// TIA Portal V19 export
FUNCTION_BLOCK "AccRollConveyor_FB"   // FB162, LAD
TITLE = Acc roll conveyor
// stored: MemoryReserve 100, SetENOAutomatically false
   VAR_INPUT
      AreaInterface : "AreaInterface";
      ZSI : "udt_ZoneSafetyInterface";
      DSI : Struct
         Roll1 : "udt_DeviceSafetyInterface";
         Roll2 : "udt_DeviceSafetyInterface";
         Roll3 : "udt_DeviceSafetyInterface";
         PusherVert : "udt_DeviceSafetyInterface";
         PusherHoriz : "udt_DeviceSafetyInterface";
      END_STRUCT;
      Drive : Struct
         Roll1 : "TAx_DriveInterface";
         Roll2 : "TAx_DriveInterface";
         Roll3 : "TAx_DriveInterface";
      END_STRUCT;
      HWID : Struct
         Roll1_TEL1 : HW_SUBMODULE;
         Roll2_TEL1 : HW_SUBMODULE;
         Roll3_TEL1 : HW_SUBMODULE;
      END_STRUCT;
      DataIn : Struct
         Pb_Semiauto : Bool;
         Rolls_PbFwd : Bool;
         Rolls_PbBwd : Bool;
         PusherVert_PbUp : Bool;
         PusherVert_PbDown : Bool;
         PusherHoriz_PbLeft : Bool;
         PusherHoriz_PbRight : Bool;
         SensorMatPresence_S2_Entry : Bool;
         SensorMatPresence_S3 : Bool;
         SensorMatPresence_S4 : Bool;
         SensorMatPresence_S5_Stop : Bool;
         ExitLeft_MatPresence1 : Bool;
         ExitLeft_MatPresence2 : Bool;
         ExitLeft_MatPresence3 : Bool;
         ExitLeft_MatPresence4 : Bool;
      END_STRUCT;
      CIn : Struct
         Manager : Struct
            EnableStopDoorOpeningReq : Bool;
            EnableStopInPhase : Bool;
            EnableStopProgrammed : Bool;
         END_STRUCT;
         Semiautomatic : Bool;
         A03_CanLoadPiece : Bool;
         A03_InCycle : Bool;
         ReqFwdFromCut : Bool;
         StopCheckQuality : Bool;
      END_STRUCT;
      Config : Struct
         Roll1 : "SpeedMachine_Config";
         Roll2 : "SpeedMachine_Config";
         Roll3 : "SpeedMachine_Config";
         PusherVert : Array[1..6] of "ValveMachine_Config";
         PusherHoriz : Array[1..6] of "ValveMachine_Config";
         SensorsDelayOn : Time := T#100ms;
         SensorsDelayOff : Time := T#100ms;
         ExitLeftDelayOn : Time := T#100ms;
         ExitLeftDelayOff : Time := T#100ms;
      END_STRUCT;
   END_VAR
   VAR_OUTPUT
      MachineInterface : "MachineInterface";
      COut : Struct
         Rolls : Struct
            Infeed_ReqON : Bool;
            Bwd_CheckNext : Bool;
            Fwd_CheckNext : Bool;
            Standstill : Bool;
         END_STRUCT;
         PusherVert : Struct
            Rest_CheckNext : Bool;
            Work_CheckNext : Bool;
            AllStandstill : Bool;
            TwoUp : Bool;
            AllDown : Bool;
         END_STRUCT;
         PusherHoriz : Struct
            Left_CheckNext : Bool;
            Right_CheckNext : Bool;
            AllStandstill : Bool;
            InLeftPos : Bool;
            InRightPos : Bool;
         END_STRUCT;
         Manager : "udt_AccRollConveyor_COut_Manager";
      END_STRUCT;
   END_VAR
   VAR_IN_OUT
      Pers : "udt_AccRollConveyor_Pers";
   END_VAR
   VAR
      Sts : Struct
         Semiautomatic : Bool;
         OP_CanMoveFreely : Bool;
         NextTargetPathLeft : Bool;
         NextTargetPathRight : Bool;
         ActTargetPathLeft : Bool;
         ActTargetPathRight : Bool;
         TrkExitLeftFull : Bool;
         TrkPieceInRolls : Int;
         TrkPieceToCheckInRoll : Int;
         TrkPieceInLenght : LReal;
         TrkPieceRecondGoodFind : Int;
         StopCutCheckPiece : Bool;
         Pusher : Struct
            InLeftPos : Bool;
            InRightPos : Bool;
            UsedInLeftPos : Bool;
            UsedInRightPos : Bool;
            AllDown : Bool;
            TwoUp : Bool;
            Used : Array[1.."MAX_PUSHER"] of Bool;
         END_STRUCT;
         CycleTime : Struct
            PusherHoriz : Struct
               DT_W_Start : DTL;
               DT_W_Stop : DTL;
               DT_R_Start : DTL;
               DT_R_Stop : DTL;
               R_To_W_Exe : Bool;
               W_To_R_Exe : Bool;
               R_To_W_Items : Int;
               R_To_W_Sum : Time;
               W_To_R_Items : Int;
               W_To_R_Sum : Time;
            END_STRUCT;
            PPrf_PrgNoSave : DInt;
         END_STRUCT;
      END_STRUCT;
      Ctrl : Struct
         StopInPhase : Bool;
         StopProgrammed : Bool;
         Pb_Semiauto : Bool;
         Rolls : Struct
            Man_Fwd : Bool;
            Man_Bwd : Bool;
            Aut_SlowDown : Bool;
            Aut_Fwd : Bool;
            Vel : LReal;
            Entry_Vel : LReal;
            Acc : LReal;
            Dec : LReal;
         END_STRUCT;
         Pusher : Struct
            Man_Left : Bool;
            Man_Right : Bool;
            Man_Up : Bool;
            Man_Down : Bool;
            Aut_Left : Bool;
            Aut_Right : Bool;
            Aut_Up : Bool;
            Aut_Down : Bool;
         END_STRUCT;
         Cycle : Struct
            ReqNextMovePieceToLeft : Bool;
            ReqNextMovePieceToRight : Bool;
            ExeNextMovePieceToLeft : Bool;
            ExeNextMovePieceToRight : Bool;
            ReqMovePieceToLeft : Bool;
            ReqMovePieceToRight : Bool;
            ExeMovePieceToLeft : Bool;
            ExeMovePieceToRight : Bool;
         END_STRUCT;
      END_STRUCT;
      Alarm : Struct
         Roll1 : "SpeedMachine_Alr";
         Roll2 : "SpeedMachine_Alr";
         Roll3 : "SpeedMachine_Alr";
         PusherVert : Array[1.."MAX_PUSHER"] of "ValveAlr";
         PusherHoriz : Array[1.."MAX_PUSHER"] of "ValveAlr";
         TrkCloggedLeftExit : Bool;
         TrkCloggedRightA03 : Bool;
         TrkCloggedRollway : Bool;
         TrkWrongMismatch_P0 : Bool;
         TrkExitFullToChek : Bool;
      END_STRUCT;
      Warning : Struct
         Roll1 : "SpeedMachine_Wng";
         Roll2 : "SpeedMachine_Wng";
         Roll3 : "SpeedMachine_Wng";
         PusherVert : Array[1.."MAX_PUSHER"] of "ValveMachine_Wng";
         PusherHoriz : Array[1.."MAX_PUSHER"] of "ValveMachine_Wng";
      END_STRUCT;
      HMI : Struct
         PusherHoriz : Struct
            Last_R_to_W_ID : DInt;
            Last_R_to_W_Time : Time;
            Last_W_to_R_ID : DInt;
            Last_W_to_R_Time : Time;
            Avg_R_to_W_Time : Time;
            Avg_W_to_R_Time : Time;
            Avg_CycleTime_S : LReal;
            Buffer_R_to_W_Time : Array[1..#BUFFER_ITEMS] of Struct
               ID : DInt;
               Value : Time;
            END_STRUCT;
            Buffer_W_to_R_Time : Array[1..#BUFFER_ITEMS] of Struct
               ID : DInt;
               Value : Time;
            END_STRUCT;
         END_STRUCT;
      END_STRUCT;
      Roll1 : "SpeedMachine_FB";
      Roll2 : "SpeedMachine_FB";
      Roll3 : "SpeedMachine_FB";
      PusherVert : Array[1.."MAX_PUSHER"] of "ValveMachine_FB";
      PusherHoriz : Array[1.."MAX_PUSHER"] of "ValveMachine_FB";
      MatPresence_S2_Entry : "DelayOnOff_R";
      MatPresence_S3 : "DelayOnOff_R";
      MatPresence_S4 : "DelayOnOff_R";
      MatPresence_S5_Stop : "DelayOnOff_R";
      MatPresence_ExitLeft1 : "DelayOnOff_R";
      MatPresence_ExitLeft2 : "DelayOnOff_R";
      MatPresence_ExitLeft3 : "DelayOnOff_R";
      MatPresence_ExitLeft4 : "DelayOnOff_R";
      tonSlowDownRolls { S7_SetPoint := 'True'} : TON_TIME;
      tonStopRollformer : TON_TIME;
      tonSlowDownRollformer : TON_TIME;
      tonTrkMismatcP0 { S7_SetPoint := 'True'} : TON_TIME;
      Rollway_Control : "Rulliera_Control_FB";
      AUX : Struct
         Pb_Semiauto { ExternalAccessible := 'False'; ExternalVisible := 'False'; ExternalWritable := 'False'} : Bool;
         Rolls_PbFwd : Bool;
         Rolls_PbBwd : Bool;
         PusherVert_PbUp : Bool;
         PusherVert_PbDopwn : Bool;
         PusherHoriz_PbLeft : Bool;
         PusherHoriz_PbRight : Bool;
         NE_MatPresence2_Entry { ExternalAccessible := 'False'; ExternalVisible := 'False'; ExternalWritable := 'False'} : Bool;
         PE_MatPresence3 : Bool;
         PE_MatPresence5_Stop : Bool;
         PE_SlowDownRolls : Bool;
         NE_SlowDownDone : Bool;
         PusherHoriz_InLeftPos : Bool;
         PusherHoriz_InRightPos : Bool;
      END_STRUCT;
      PusherVert_MachineInterface { ExternalAccessible := 'False'; ExternalVisible := 'False'; ExternalWritable := 'False'} : "MachineInterface";
      PusherHoriz_MachineInterface { ExternalAccessible := 'False'; ExternalVisible := 'False'; ExternalWritable := 'False'} : "MachineInterface";
   END_VAR
   VAR_TEMP
      PE : Struct
         Pb_Semiauto : Bool;
         Rolls_PbFwd : Bool;
         Rolls_PbBwd : Bool;
         PusherVert_PbUp : Bool;
         PusherVert_PbDown : Bool;
         PusherHoriz_PbLeft : Bool;
         PusherHoriz_PbRight : Bool;
         NE_MatPresence2_Entry : Bool;
         PE_MatPresence3 : Bool;
         PE_MatPresence5_Stop : Bool;
         PE_SlowDownRolls : Bool;
         NE_SlowDownDone : Bool;
         PusherHoriz_InLeftPos : Bool;
         PusherHoriz_InRightPos : Bool;
      END_STRUCT;
      i : Int;
      PusherVert_NrUp : Int;
      ActualPieceLenght : LReal;
      RetVal_MOVEBLK : Int;
      Ptrk_ItemFind : Int;
      Ptrk_ExitItemToCheck : Int;
      ReturnVal : Word;
      AddAlarm : Bool;
      PartLenght : LReal;
   END_VAR
   VAR CONSTANT
      BUFFER_ITEMS : Int := 10;
   END_VAR
   VAR_TEMP   // added for the SCL form of the ladder/FBD networks
      _w1 : Bool;
      _w2 : Bool;
      _w3 : Bool;
      _w4 : Bool;
      _w5 : Bool;
   END_VAR
BEGIN

REGION Network 1 (SCL): Reset alarms command

   IF  #AreaInterface.RstAlarms THEN
       // Alarms
       #Alarm.TrkCloggedLeftExit := FALSE;
       #Alarm.TrkCloggedRightA03 := FALSE;
       #Alarm.TrkCloggedRollway := FALSE;

       #Alarm.TrkWrongMismatch_P0 := FALSE;
       #Alarm.TrkExitFullToChek := FALSE;

   END_IF;
END_REGION

REGION Network 2: >
END_REGION

REGION Network 3: OP Can move freely
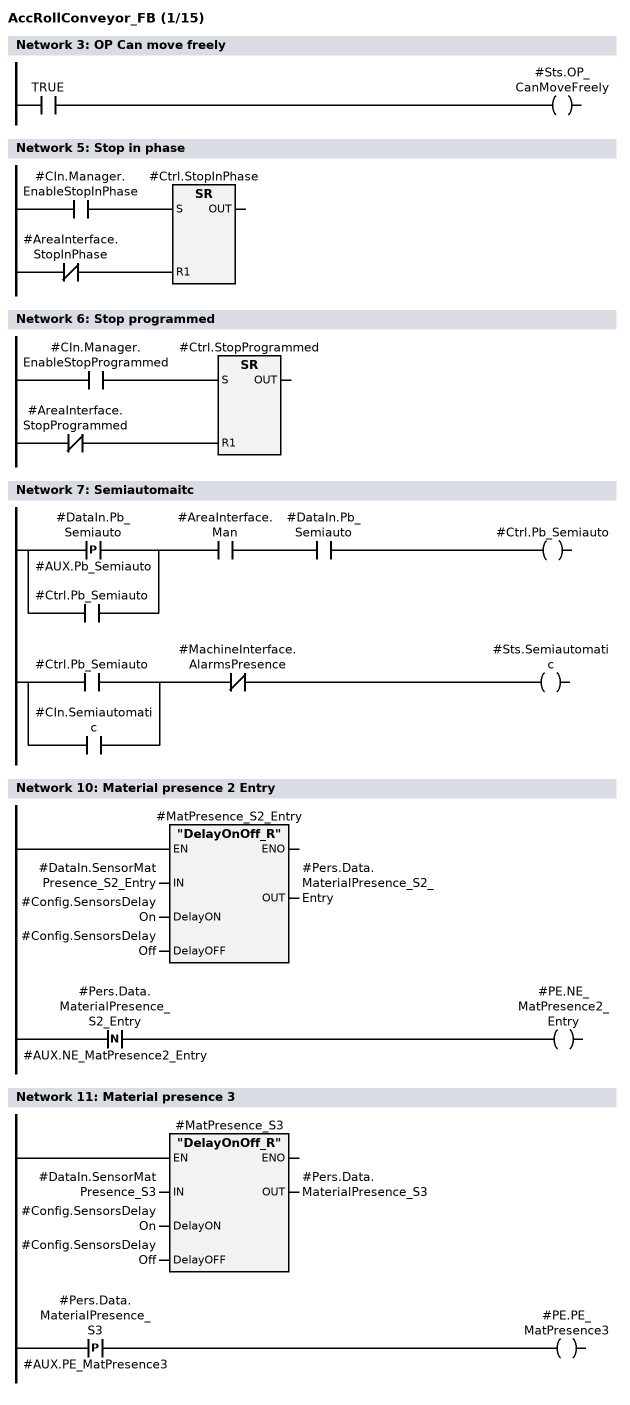
   RUNG wire#powerrail
      Contact( TRUE )
      Coil( #Sts.OP_CanMoveFreely )
   END_RUNG
   // the same network as SCL:
   #Sts.OP_CanMoveFreely := TRUE;
END_REGION

REGION Network 5: Stop in phase
   RUNG wire#powerrail
      Contact( #CIn.Manager.EnableStopInPhase )
      S_SR(operand := #Ctrl.StopInPhase, r1 := wire#w1)
   END_RUNG
   RUNG wire#powerrail
      I_Contact( #AreaInterface.StopInPhase )
   END_RUNG wire#w1
   // the same network as SCL:
   IF #CIn.Manager.EnableStopInPhase THEN
       #Ctrl.StopInPhase := TRUE;   // SR flip-flop
   END_IF;
   IF NOT #AreaInterface.StopInPhase THEN #Ctrl.StopInPhase := FALSE; END_IF;
END_REGION

REGION Network 6: Stop programmed
   RUNG wire#powerrail
      Contact( #CIn.Manager.EnableStopProgrammed )
      S_SR(operand := #Ctrl.StopProgrammed, r1 := wire#w1)
   END_RUNG
   RUNG wire#powerrail
      I_Contact( #AreaInterface.StopProgrammed )
   END_RUNG wire#w1
   // the same network as SCL:
   IF #CIn.Manager.EnableStopProgrammed THEN
       #Ctrl.StopProgrammed := TRUE;   // SR flip-flop
   END_IF;
   IF NOT #AreaInterface.StopProgrammed THEN #Ctrl.StopProgrammed := FALSE; END_IF;
END_REGION

REGION Network 7: Semiautomaitc
   RUNG wire#powerrail
      P_Contact(operand := #DataIn.Pb_Semiauto, bit := #AUX.Pb_Semiauto)
      wire#w1
      Contact( #AreaInterface.Man )
      Contact( #DataIn.Pb_Semiauto )
      Coil( #Ctrl.Pb_Semiauto )
   END_RUNG
   RUNG wire#powerrail
      Contact( #Ctrl.Pb_Semiauto )
   END_RUNG wire#w1
   RUNG wire#powerrail
      Contact( #Ctrl.Pb_Semiauto )
      wire#w2
      I_Contact( #MachineInterface.AlarmsPresence )
      Coil( #Sts.Semiautomatic )
   END_RUNG
   RUNG wire#powerrail
      Contact( #CIn.Semiautomatic )
   END_RUNG wire#w2
   // the same network as SCL:
   #_w1 := #DataIn.Pb_Semiauto AND NOT #AUX.Pb_Semiauto;   // rising edge of #DataIn.Pb_Semiauto
   #AUX.Pb_Semiauto := #DataIn.Pb_Semiauto;
   #Ctrl.Pb_Semiauto := (#_w1 OR #Ctrl.Pb_Semiauto) AND #AreaInterface.Man AND #DataIn.Pb_Semiauto;
   #Sts.Semiautomatic := (#Ctrl.Pb_Semiauto OR #CIn.Semiautomatic) AND NOT #MachineInterface.AlarmsPresence;
END_REGION

REGION Network 9: <<< SENSOR MAT PRESENCE >>>
END_REGION

REGION Network 10: Material presence 2 Entry
   RUNG wire#powerrail
      #MatPresence_S2_Entry(IN := #DataIn.SensorMatPresence_S2_Entry, DelayON := #Config.SensorsDelayOn, DelayOFF := #Config.SensorsDelayOff, OUT => #Pers.Data.MaterialPresence_S2_Entry)
   END_RUNG
   RUNG wire#powerrail
      N_Contact(operand := #Pers.Data.MaterialPresence_S2_Entry, bit := #AUX.NE_MatPresence2_Entry)
      Coil( #PE.NE_MatPresence2_Entry )
   END_RUNG
   // the same network as SCL:
   #MatPresence_S2_Entry(IN := #DataIn.SensorMatPresence_S2_Entry,   // "DelayOnOff_R"
                         DelayON := #Config.SensorsDelayOn,
                         DelayOFF := #Config.SensorsDelayOff,
                         OUT => #Pers.Data.MaterialPresence_S2_Entry);
   #_w1 := NOT #Pers.Data.MaterialPresence_S2_Entry AND #AUX.NE_MatPresence2_Entry;   // falling edge of #Pers.Data.MaterialPresence_S2_Entry
   #AUX.NE_MatPresence2_Entry := #Pers.Data.MaterialPresence_S2_Entry;
   #PE.NE_MatPresence2_Entry := #_w1;
END_REGION

REGION Network 11: Material presence 3
   RUNG wire#powerrail
      #MatPresence_S3(IN := #DataIn.SensorMatPresence_S3, DelayON := #Config.SensorsDelayOn, DelayOFF := #Config.SensorsDelayOff, OUT => #Pers.Data.MaterialPresence_S3)
   END_RUNG
   RUNG wire#powerrail
      P_Contact(operand := #Pers.Data.MaterialPresence_S3, bit := #AUX.PE_MatPresence3)
      Coil( #PE.PE_MatPresence3 )
   END_RUNG
   // the same network as SCL:
   #MatPresence_S3(IN := #DataIn.SensorMatPresence_S3,   // "DelayOnOff_R"
                   DelayON := #Config.SensorsDelayOn,
                   DelayOFF := #Config.SensorsDelayOff,
                   OUT => #Pers.Data.MaterialPresence_S3);
   #_w1 := #Pers.Data.MaterialPresence_S3 AND NOT #AUX.PE_MatPresence3;   // rising edge of #Pers.Data.MaterialPresence_S3
   #AUX.PE_MatPresence3 := #Pers.Data.MaterialPresence_S3;
   #PE.PE_MatPresence3 := #_w1;
END_REGION

REGION Network 12: Material presence 4
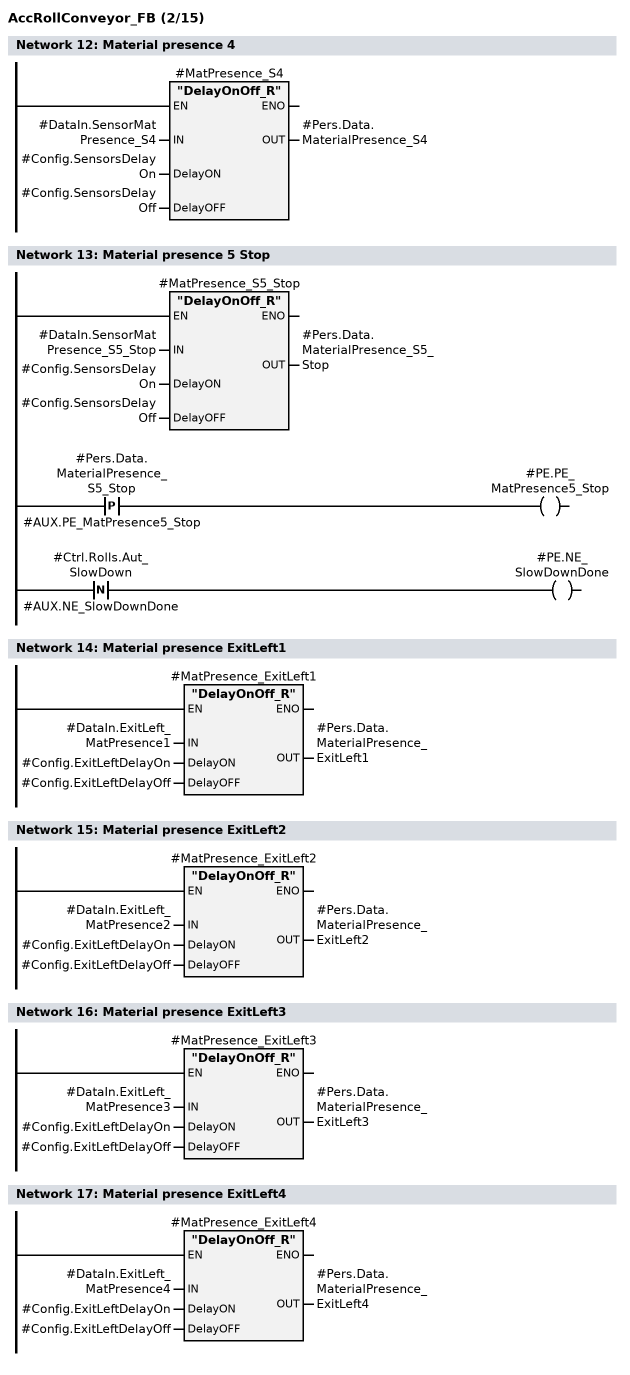
   RUNG wire#powerrail
      #MatPresence_S4(IN := #DataIn.SensorMatPresence_S4, DelayON := #Config.SensorsDelayOn, DelayOFF := #Config.SensorsDelayOff, OUT => #Pers.Data.MaterialPresence_S4)
   END_RUNG
   // the same network as SCL:
   #MatPresence_S4(IN := #DataIn.SensorMatPresence_S4,   // "DelayOnOff_R"
                   DelayON := #Config.SensorsDelayOn,
                   DelayOFF := #Config.SensorsDelayOff,
                   OUT => #Pers.Data.MaterialPresence_S4);
END_REGION

REGION Network 13: Material presence 5 Stop
   RUNG wire#powerrail
      #MatPresence_S5_Stop(IN := #DataIn.SensorMatPresence_S5_Stop, DelayON := #Config.SensorsDelayOn, DelayOFF := #Config.SensorsDelayOff, OUT => #Pers.Data.MaterialPresence_S5_Stop)
   END_RUNG
   RUNG wire#powerrail
      P_Contact(operand := #Pers.Data.MaterialPresence_S5_Stop, bit := #AUX.PE_MatPresence5_Stop)
      Coil( #PE.PE_MatPresence5_Stop )
   END_RUNG
   RUNG wire#powerrail
      N_Contact(operand := #Ctrl.Rolls.Aut_SlowDown, bit := #AUX.NE_SlowDownDone)
      Coil( #PE.NE_SlowDownDone )
   END_RUNG
   // the same network as SCL:
   #MatPresence_S5_Stop(IN := #DataIn.SensorMatPresence_S5_Stop,   // "DelayOnOff_R"
                        DelayON := #Config.SensorsDelayOn,
                        DelayOFF := #Config.SensorsDelayOff,
                        OUT => #Pers.Data.MaterialPresence_S5_Stop);
   #_w1 := #Pers.Data.MaterialPresence_S5_Stop AND NOT #AUX.PE_MatPresence5_Stop;   // rising edge of #Pers.Data.MaterialPresence_S5_Stop
   #AUX.PE_MatPresence5_Stop := #Pers.Data.MaterialPresence_S5_Stop;
   #PE.PE_MatPresence5_Stop := #_w1;
   #_w2 := NOT #Ctrl.Rolls.Aut_SlowDown AND #AUX.NE_SlowDownDone;   // falling edge of #Ctrl.Rolls.Aut_SlowDown
   #AUX.NE_SlowDownDone := #Ctrl.Rolls.Aut_SlowDown;
   #PE.NE_SlowDownDone := #_w2;
END_REGION

REGION Network 14: Material presence ExitLeft1
   RUNG wire#powerrail
      #MatPresence_ExitLeft1(IN := #DataIn.ExitLeft_MatPresence1, DelayON := #Config.ExitLeftDelayOn, DelayOFF := #Config.ExitLeftDelayOff, OUT => #Pers.Data.MaterialPresence_ExitLeft1)
   END_RUNG
   // the same network as SCL:
   #MatPresence_ExitLeft1(IN := #DataIn.ExitLeft_MatPresence1,   // "DelayOnOff_R"
                          DelayON := #Config.ExitLeftDelayOn,
                          DelayOFF := #Config.ExitLeftDelayOff,
                          OUT => #Pers.Data.MaterialPresence_ExitLeft1);
END_REGION

REGION Network 15: Material presence ExitLeft2
   RUNG wire#powerrail
      #MatPresence_ExitLeft2(IN := #DataIn.ExitLeft_MatPresence2, DelayON := #Config.ExitLeftDelayOn, DelayOFF := #Config.ExitLeftDelayOff, OUT => #Pers.Data.MaterialPresence_ExitLeft2)
   END_RUNG
   // the same network as SCL:
   #MatPresence_ExitLeft2(IN := #DataIn.ExitLeft_MatPresence2,   // "DelayOnOff_R"
                          DelayON := #Config.ExitLeftDelayOn,
                          DelayOFF := #Config.ExitLeftDelayOff,
                          OUT => #Pers.Data.MaterialPresence_ExitLeft2);
END_REGION

REGION Network 16: Material presence ExitLeft3
   RUNG wire#powerrail
      #MatPresence_ExitLeft3(IN := #DataIn.ExitLeft_MatPresence3, DelayON := #Config.ExitLeftDelayOn, DelayOFF := #Config.ExitLeftDelayOff, OUT => #Pers.Data.MaterialPresence_ExitLeft3)
   END_RUNG
   // the same network as SCL:
   #MatPresence_ExitLeft3(IN := #DataIn.ExitLeft_MatPresence3,   // "DelayOnOff_R"
                          DelayON := #Config.ExitLeftDelayOn,
                          DelayOFF := #Config.ExitLeftDelayOff,
                          OUT => #Pers.Data.MaterialPresence_ExitLeft3);
END_REGION

REGION Network 17: Material presence ExitLeft4
   RUNG wire#powerrail
      #MatPresence_ExitLeft4(IN := #DataIn.ExitLeft_MatPresence4, DelayON := #Config.ExitLeftDelayOn, DelayOFF := #Config.ExitLeftDelayOff, OUT => #Pers.Data.MaterialPresence_ExitLeft4)
   END_RUNG
   // the same network as SCL:
   #MatPresence_ExitLeft4(IN := #DataIn.ExitLeft_MatPresence4,   // "DelayOnOff_R"
                          DelayON := #Config.ExitLeftDelayOn,
                          DelayOFF := #Config.ExitLeftDelayOff,
                          OUT => #Pers.Data.MaterialPresence_ExitLeft4);
END_REGION

REGION Network 18: >
END_REGION

REGION Network 19: <<< TRACKING >>>
END_REGION

REGION Network 20 (SCL): Rollway movement

   //Tracking ENTRY to P6 
   IF "PTrk".A0202.P[PTRK_A0202_ENTRY].P_ID <> 0 AND
       ((#PE.NE_MatPresence2_Entry AND "PTrk".A0202.P[PTRK_A0202_ENTRY].PLen_Meas <= 4000) OR
       (#Pers.Data.MaterialPresence_S3 AND "PTrk".A0202.P[PTRK_A0202_ENTRY].PLen_Meas > 4000))
   THEN
       IF "PTrk".A0202.P[PTRK_A0202_P6].P_ID = 0 THEN
           "PTrk".A0202.P[PTRK_A0202_P6] := "PTrk".A0202.P[PTRK_A0202_ENTRY];
           "PTrk".A0202.P[PTRK_A0202_ENTRY] := "PTrk".Empty;
       ELSE
           #Alarm.TrkCloggedRollway := TRUE;
       END_IF;

   END_IF;


   //Sposto buffer tacking
   #i := "PTRK_A0202_P1";
   WHILE #i > "PTRK_A0202_P6" DO

       IF "PTrk".A0202.P[#i].P_ID = 0 AND
           "PTrk".A0202.P[#i - 1].P_ID <> 0
       THEN
           "PTrk".A0202.P[#i] := "PTrk".A0202.P[#i - 1];
           "PTrk".A0202.P[#i - 1] := "PTrk".Empty;
       END_IF;
       #i -= 1;

   END_WHILE;


   //Tracking P1 to P0
   IF "PTrk".A0202.P[PTRK_A0202_P1].P_ID <> 0 AND
       ((#PE.PE_MatPresence5_Stop AND #AreaInterface.Man AND NOT #Sts.Semiautomatic)
         OR #PE.NE_SlowDownDone)
   THEN
       IF "PTrk".A0202.P[PTRK_A0202_P0].P_ID = 0 THEN
           "PTrk".A0202.P[PTRK_A0202_P0] := "PTrk".A0202.P[PTRK_A0202_P1];
           "PTrk".A0202.P[PTRK_A0202_P1] := "PTrk".Empty;
       ELSE
           #Alarm.TrkCloggedRollway := TRUE;
       END_IF;
   END_IF;
END_REGION

REGION Network 21 (SCL): Left Exit movement

   //Rollway to left
   IF "PTrk".A0202.P[PTRK_A0202_P0].P_ID <> 0 AND
       (#Ctrl.Cycle.ReqMovePieceToLeft OR #AreaInterface.Man) AND
       #COut.PusherHoriz.Left_CheckNext AND NOT #COut.PusherHoriz.AllStandstill AND
       #Sts.Pusher.TwoUp AND
       NOT #Sts.Pusher.InLeftPos
   THEN

       IF "PTrk".A0202.P[PTRK_A0202_DEVITATOR_To_EXIT].P_ID = 0  THEN
           "PTrk".A0202.P[PTRK_A0202_DEVITATOR_To_EXIT] := "PTrk".A0202.P[PTRK_A0202_P0];
           "PTrk".A0202.P[PTRK_A0202_P0] := "PTrk".Empty;
       ELSE
           #Alarm.TrkCloggedLeftExit := TRUE;
       END_IF;
   END_IF;

   //Left to Exit
   IF "PTrk".A0202.P[PTRK_A0202_DEVITATOR_To_EXIT].P_ID <> 0 AND
       #Sts.Pusher.TwoUp AND
       #Sts.Pusher.UsedInLeftPos
   THEN

       #RetVal_MOVEBLK := MOVE_BLK_VARIANT(SRC := "PTrk".A02_EXIT_TOCHECK,
                                           COUNT := INT_TO_UDINT("PTRK_A0202_EXIT_TOCHECK_ITEMS" - 1),
                                           SRC_INDEX := 0,
                                           DEST_INDEX := 1,
                                           DEST => "PTrk".A02_EXIT_TOCHECK);

       "PTrk".A02_EXIT_TOCHECK[1] := "PTrk".A0202.P[PTRK_A0202_DEVITATOR_To_EXIT];
       "PTrk".A0202.P[PTRK_A0202_DEVITATOR_To_EXIT] := "PTrk".Empty;
   END_IF;

   //Alarm Clogged
   IF "PTrk".A0202.P[PTRK_A0202_DEVITATOR_To_EXIT].P_ID <> 0 AND
        "PTrk".A0202.P[PTRK_A0202_P0].P_ID <> 0
   THEN
       #Alarm.TrkCloggedLeftExit := TRUE;
   END_IF;
END_REGION

REGION Network 22 (SCL): Right A03 movement

   //Rollway to left
   IF "PTrk".A0202.P[PTRK_A0202_P0].P_ID <> 0 AND
       (#Ctrl.Cycle.ReqMovePieceToRight OR #AreaInterface.Man) AND
       #COut.PusherHoriz.Right_CheckNext AND NOT #COut.PusherHoriz.AllStandstill AND
       #Sts.Pusher.TwoUp AND 
       NOT #Sts.Pusher.InRightPos
   THEN

       IF "PTrk".A0202.P[PTRK_A0202_DEVIATOR_To_A0301].P_ID = 0 AND
           "PTrk".A0301.P[PTRK_A0301_Pos1_Entry].P_ID = 0
       THEN
           "PTrk".A0202.P[PTRK_A0202_DEVIATOR_To_A0301] := "PTrk".A0202.P[PTRK_A0202_P0];
           "PTrk".A0202.P[PTRK_A0202_P0] := "PTrk".Empty;
       ELSE
           #Alarm.TrkCloggedRightA03 := TRUE;
       END_IF;
   END_IF;

   //Left to Exit
   IF "PTrk".A0202.P[PTRK_A0202_DEVIATOR_To_A0301].P_ID <> 0 AND
       #Sts.Pusher.TwoUp AND
       #Sts.Pusher.UsedInRightPos
   THEN
       "PTrk".A0301.P[PTRK_A0301_Pos1_Entry] := "PTrk".A0202.P[PTRK_A0202_DEVIATOR_To_A0301];
       "PTrk".A0202.P[PTRK_A0202_DEVIATOR_To_A0301] := "PTrk".Empty;
   END_IF;

   //Alarm Clogged
   IF "PTrk".A0202.P[PTRK_A0202_DEVIATOR_To_A0301].P_ID <> 0 AND
       ("PTrk".A0301.P[PTRK_A0301_Pos1_Entry].P_ID <> 0 OR "PTrk".A0202.P[PTRK_A0202_P0].P_ID <> 0)
   THEN
       #Alarm.TrkCloggedRightA03 := TRUE;
   END_IF;
END_REGION

REGION Network 23 (SCL): Exit To check manager

   //Shift verso alto se trovo buco

   #Ptrk_ItemFind := 0;
   FOR #i := 1 TO "PTRK_A0202_EXIT_TOCHECK_ITEMS" - 1 DO

       IF "PTrk".A02_EXIT_TOCHECK[#i].P_ID = 0 AND
           "PTrk".A02_EXIT_TOCHECK[#i + 1].P_ID <> 0 THEN
           #Ptrk_ItemFind := #i;
           EXIT;
       END_IF;
   END_FOR;

   IF #Ptrk_ItemFind > 0 THEN
       #RetVal_MOVEBLK := MOVE_BLK_VARIANT(SRC := "PTrk".A02_EXIT_TOCHECK,
                                           COUNT := INT_TO_UDINT("PTRK_A0202_EXIT_TOCHECK_ITEMS" - #Ptrk_ItemFind),
                                           SRC_INDEX := #Ptrk_ItemFind,
                                           DEST_INDEX := #Ptrk_ItemFind - 1,
                                           DEST => "PTrk".A02_EXIT_TOCHECK);
   END_IF;



   //Conteggio Pezzi su rulliera
   #Sts.TrkPieceInRolls := 0;
   #Sts.TrkPieceInLenght := 0.0;
   #Sts.TrkPieceToCheckInRoll := 0;

   FOR #i := 1 TO "PTRK_A0202_DEVITATOR_To_EXIT" DO

       IF "PTrk".A0202.P[#i].P_ID <> 0 THEN
           #Sts.TrkPieceInRolls += 1;
           #Sts.TrkPieceInLenght := "PTrk".A0202.P[#i].PLen_Meas;

           //Conto i pezzi da controllare
           IF "PTrk".A0202.P[#i].Quality = "TO_CHECK" OR
               "PTrk".A0202.P[#i].Quality = "TO_CHECK_LEN"
           THEN
               #Sts.TrkPieceToCheckInRoll += 1;
           END_IF;

       END_IF;

   END_FOR;

   //Rulliera vuota
   #COut.Manager.Empty := #Sts.TrkPieceInRolls = 0;


   //Rallentamento profila se pezzi da controllare
   #Ptrk_ExitItemToCheck := "PTRK_A0202_EXIT_TOCHECK_ITEMS" - #Sts.TrkPieceToCheckInRoll;
   IF #Ptrk_ExitItemToCheck < 1 THEN
       #Ptrk_ExitItemToCheck := 1;
   END_IF;


   #Sts.StopCutCheckPiece := FALSE;
   #Sts.TrkPieceRecondGoodFind := 0;
   FOR #i := 1 TO "PTRK_A0202_EXIT_TOCHECK_ITEMS" DO

       IF #i >= #Ptrk_ExitItemToCheck AND
           "PTrk".A02_EXIT_TOCHECK[#i].P_ID <> 0 AND
           ("PTrk".A02_EXIT_TOCHECK[#i].Quality = "TO_CHECK" OR
           "PTrk".A02_EXIT_TOCHECK[#i].Quality = "TO_CHECK_LEN")
       THEN
           #Sts.StopCutCheckPiece := TRUE;
       END_IF;

       IF "PTrk".A02_EXIT_TOCHECK[#i].P_ID <> 0
           AND "PTrk".A02_EXIT_TOCHECK[#i].Quality = "RECOND_GOOD"
       THEN
           #Sts.TrkPieceRecondGoodFind := #i;
       END_IF;
   END_FOR;


   //Move piece recond good
   IF #Sts.TrkPieceRecondGoodFind > 0 AND
       "PTrk".A0202.P[PTRK_A0202_P0].P_ID = 0
   THEN
       "PTrk".A0202.P[PTRK_A0202_P0] := "PTrk".A02_EXIT_TOCHECK[#Sts.TrkPieceRecondGoodFind];
   END_IF;




   //Tracking left FULL
   #Sts.TrkExitLeftFull :=
   ("PTrk".A02_EXIT_TOCHECK[PTRK_A0202_EXIT_TOCHECK_ITEMS].P_ID <> 0 AND "PTrk".A02_EXIT_TOCHECK[PTRK_A0202_EXIT_TOCHECK_ITEMS].Quality = "TO_CHECK") OR
   ("PTrk".A02_EXIT_TOCHECK[PTRK_A0202_EXIT_TOCHECK_ITEMS].P_ID <> 0 AND "PTrk".A02_EXIT_TOCHECK[PTRK_A0202_EXIT_TOCHECK_ITEMS].Quality = "TO_CHECK_LEN") OR
   ((#Pers.Data.MaterialPresence_ExitLeft3 OR #Pers.Data.MaterialPresence_ExitLeft4) AND
   (#Pers.Data.MaterialPresence_ExitLeft1 OR #Pers.Data.MaterialPresence_ExitLeft2));

   //Allarme Trk full
   IF("PTrk".A02_EXIT_TOCHECK[PTRK_A0202_EXIT_TOCHECK_ITEMS].P_ID <> 0 AND "PTrk".A02_EXIT_TOCHECK[PTRK_A0202_EXIT_TOCHECK_ITEMS].Quality = "TO_CHECK") OR
       ("PTrk".A02_EXIT_TOCHECK[PTRK_A0202_EXIT_TOCHECK_ITEMS].P_ID <> 0 AND "PTrk".A02_EXIT_TOCHECK[PTRK_A0202_EXIT_TOCHECK_ITEMS].Quality = "TO_CHECK_LEN")
   THEN
       #Alarm.TrkExitFullToChek := TRUE;
   END_IF;
END_REGION

REGION Network 24: Alarm mismatch P0
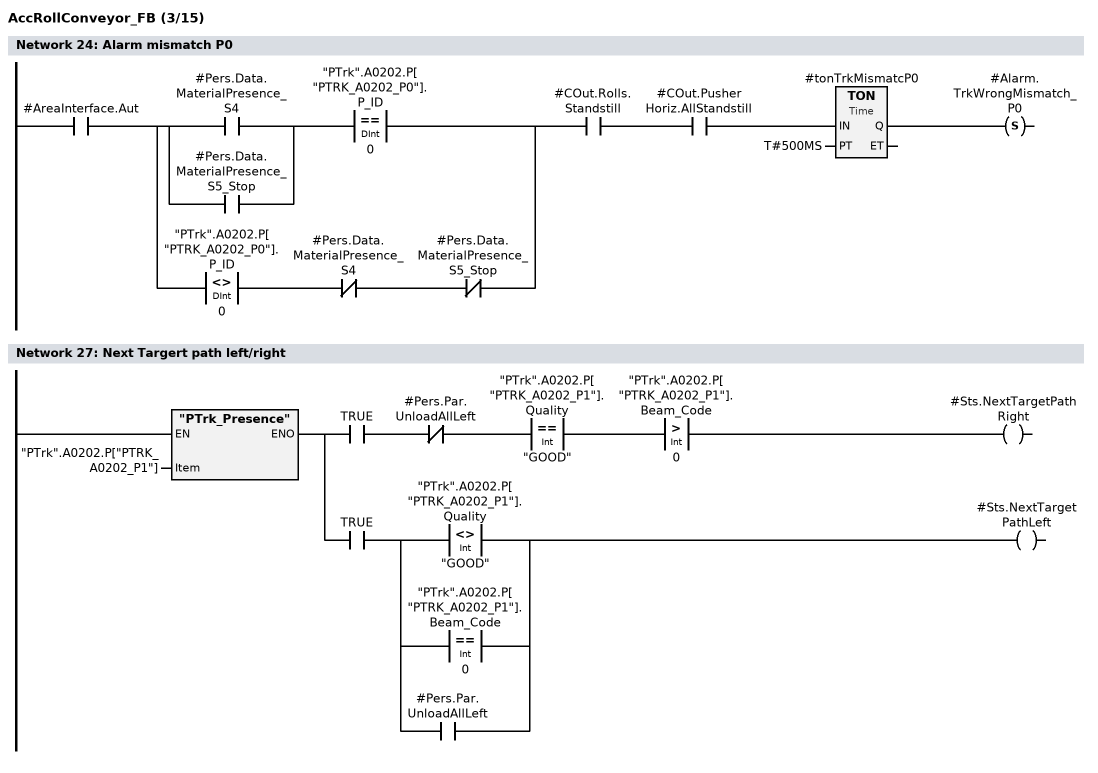
   RUNG wire#powerrail
      Contact( #AreaInterface.Aut )
      wire#w1
      Contact( #Pers.Data.MaterialPresence_S4 )
      wire#w2
      { S7_Templates := "SrcType := DInt" } EQ_Contact(in1 := "PTrk".A0202.P["PTRK_A0202_P0"].P_ID, in2 := 0)
      wire#w3
      Contact( #COut.Rolls.Standstill )
      Contact( #COut.PusherHoriz.AllStandstill )
      { S7_Templates := "time_type := Time" } #tonTrkMismatcP0.TON(pt := T#500MS, et =>)
      S_Coil( #Alarm.TrkWrongMismatch_P0 )
   END_RUNG
   RUNG wire#w1
      Contact( #Pers.Data.MaterialPresence_S5_Stop )
   END_RUNG wire#w2
   RUNG wire#w1
      { S7_Templates := "SrcType := DInt" } NE_Contact(in1 := "PTrk".A0202.P["PTRK_A0202_P0"].P_ID, in2 := 0)
      I_Contact( #Pers.Data.MaterialPresence_S4 )
      I_Contact( #Pers.Data.MaterialPresence_S5_Stop )
   END_RUNG wire#w3
   // the same network as SCL:
   #tonTrkMismatcP0(IN := #AreaInterface.Aut AND (((#Pers.Data.MaterialPresence_S4 OR #Pers.Data.MaterialPresence_S5_Stop) AND ("PTrk".A0202.P["PTRK_A0202_P0"].P_ID = 0)) OR (("PTrk".A0202.P["PTRK_A0202_P0"].P_ID <> 0) AND NOT #Pers.Data.MaterialPresence_S4 AND NOT #Pers.Data.MaterialPresence_S5_Stop)) AND #COut.Rolls.Standstill AND #COut.PusherHoriz.AllStandstill,   // TON
                    PT := T#500MS);
   IF #tonTrkMismatcP0.Q THEN #Alarm.TrkWrongMismatch_P0 := TRUE; END_IF;
END_REGION

REGION Network 25: >
END_REGION

REGION Network 26: <<<PUSHER MANGER >>>
END_REGION

REGION Network 27: Next Targert path left/right
   RUNG wire#powerrail
      "PTrk_Presence"(Item := "PTrk".A0202.P["PTRK_A0202_P1"])
      wire#w1
      Contact( TRUE )
      I_Contact( #Pers.Par.UnloadAllLeft )
      { S7_Templates := "SrcType := Int" } EQ_Contact(in1 := "PTrk".A0202.P["PTRK_A0202_P1"].Quality, in2 := "GOOD")
      { S7_Templates := "SrcType := Int" } GT_Contact(in1 := "PTrk".A0202.P["PTRK_A0202_P1"].Beam_Code, in2 := 0)
      Coil( #Sts.NextTargetPathRight )
   END_RUNG
   RUNG wire#w1
      Contact( TRUE )
      wire#w2
      { S7_Templates := "SrcType := Int" } NE_Contact(in1 := "PTrk".A0202.P["PTRK_A0202_P1"].Quality, in2 := "GOOD")
      wire#w3
      Coil( #Sts.NextTargetPathLeft )
   END_RUNG
   RUNG wire#w2
      { S7_Templates := "SrcType := Int" } EQ_Contact(in1 := "PTrk".A0202.P["PTRK_A0202_P1"].Beam_Code, in2 := 0)
   END_RUNG wire#w3
   RUNG wire#w2
      Contact( #Pers.Par.UnloadAllLeft )
   END_RUNG wire#w3
   // the same network as SCL:
   "PTrk_Presence"(Item := "PTrk".A0202.P["PTRK_A0202_P1"], ENO => #_w1);
   #Sts.NextTargetPathRight := #_w1 AND TRUE AND NOT #Pers.Par.UnloadAllLeft AND ("PTrk".A0202.P["PTRK_A0202_P1"].Quality = "GOOD") AND ("PTrk".A0202.P["PTRK_A0202_P1"].Beam_Code > 0);
   #Sts.NextTargetPathLeft := #_w1 AND TRUE AND (("PTrk".A0202.P["PTRK_A0202_P1"].Quality <> "GOOD") OR ("PTrk".A0202.P["PTRK_A0202_P1"].Beam_Code = 0) OR #Pers.Par.UnloadAllLeft);
END_REGION

REGION Network 28: Actual Targert path left/right
   // Sys.Bypass Delu il semiguscio può essere anche NG !!!
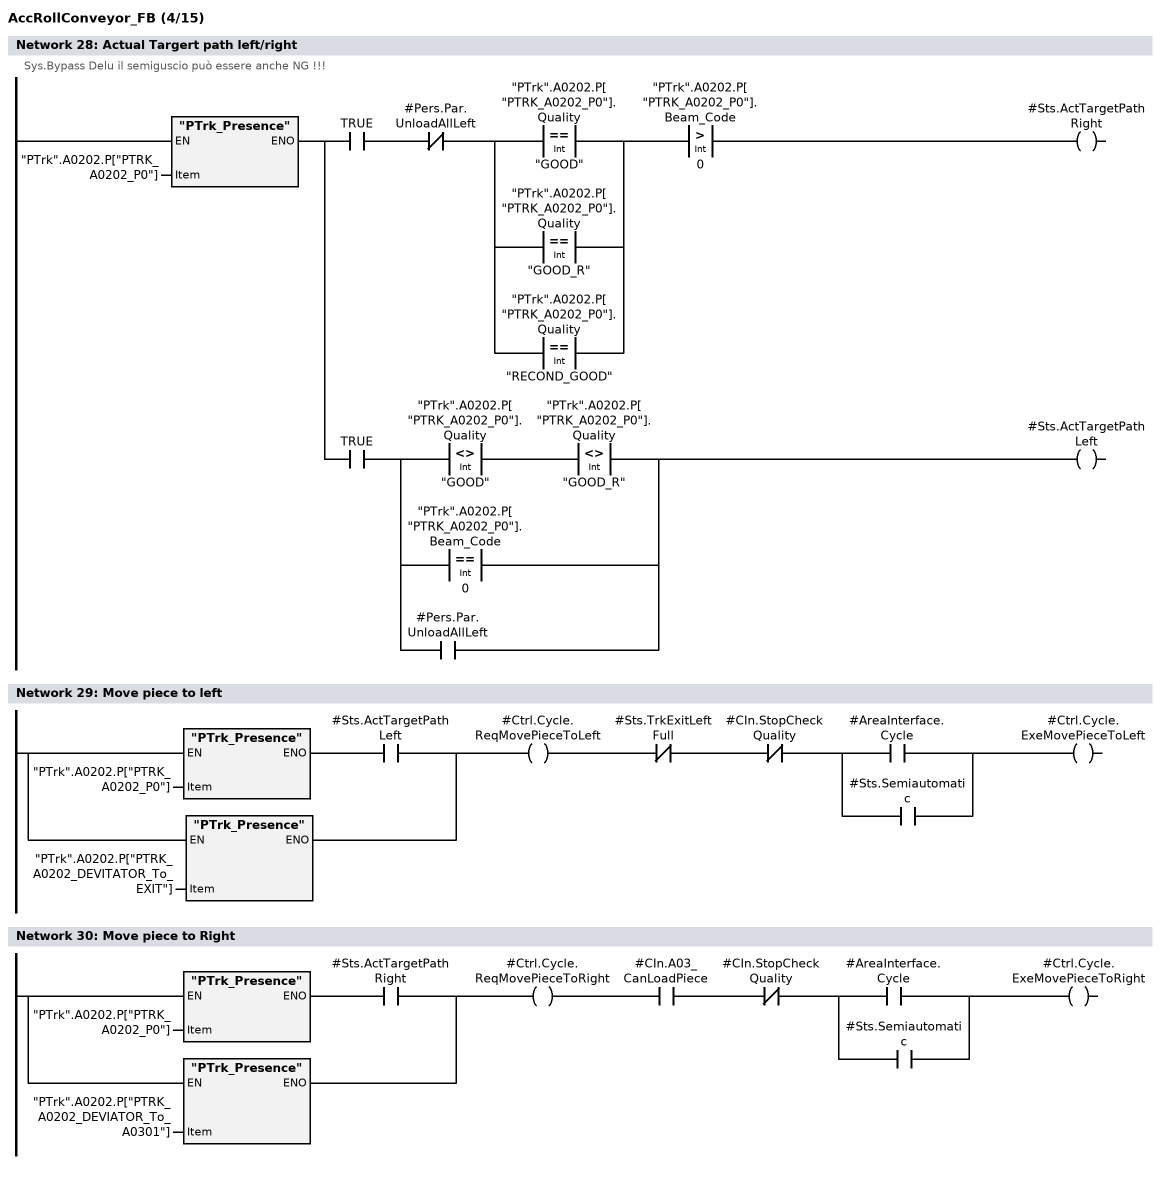
   RUNG wire#powerrail
      "PTrk_Presence"(Item := "PTrk".A0202.P["PTRK_A0202_P0"])
      wire#w1
      Contact( TRUE )
      I_Contact( #Pers.Par.UnloadAllLeft )
      wire#w2
      { S7_Templates := "SrcType := Int" } EQ_Contact(in1 := "PTrk".A0202.P["PTRK_A0202_P0"].Quality, in2 := "GOOD")
      wire#w3
      { S7_Templates := "SrcType := Int" } GT_Contact(in1 := "PTrk".A0202.P["PTRK_A0202_P0"].Beam_Code, in2 := 0)
      Coil( #Sts.ActTargetPathRight )
   END_RUNG
   RUNG wire#w2
      { S7_Templates := "SrcType := Int" } EQ_Contact(in1 := "PTrk".A0202.P["PTRK_A0202_P0"].Quality, in2 := "GOOD_R")
   END_RUNG wire#w3
   RUNG wire#w2
      { S7_Templates := "SrcType := Int" } EQ_Contact(in1 := "PTrk".A0202.P["PTRK_A0202_P0"].Quality, in2 := "RECOND_GOOD")
   END_RUNG wire#w3
   RUNG wire#w1
      Contact( TRUE )
      wire#w4
      { S7_Templates := "SrcType := Int" } NE_Contact(in1 := "PTrk".A0202.P["PTRK_A0202_P0"].Quality, in2 := "GOOD")
      { S7_Templates := "SrcType := Int" } NE_Contact(in1 := "PTrk".A0202.P["PTRK_A0202_P0"].Quality, in2 := "GOOD_R")
      wire#w5
      Coil( #Sts.ActTargetPathLeft )
   END_RUNG
   RUNG wire#w4
      { S7_Templates := "SrcType := Int" } EQ_Contact(in1 := "PTrk".A0202.P["PTRK_A0202_P0"].Beam_Code, in2 := 0)
   END_RUNG wire#w5
   RUNG wire#w4
      Contact( #Pers.Par.UnloadAllLeft )
   END_RUNG wire#w5
   // the same network as SCL:
   "PTrk_Presence"(Item := "PTrk".A0202.P["PTRK_A0202_P0"], ENO => #_w1);
   #Sts.ActTargetPathRight := #_w1 AND TRUE AND NOT #Pers.Par.UnloadAllLeft AND (("PTrk".A0202.P["PTRK_A0202_P0"].Quality = "GOOD") OR ("PTrk".A0202.P["PTRK_A0202_P0"].Quality = "GOOD_R") OR ("PTrk".A0202.P["PTRK_A0202_P0"].Quality = "RECOND_GOOD")) AND ("PTrk".A0202.P["PTRK_A0202_P0"].Beam_Code > 0);
   #Sts.ActTargetPathLeft := #_w1 AND TRUE AND ((("PTrk".A0202.P["PTRK_A0202_P0"].Quality <> "GOOD") AND ("PTrk".A0202.P["PTRK_A0202_P0"].Quality <> "GOOD_R")) OR ("PTrk".A0202.P["PTRK_A0202_P0"].Beam_Code = 0) OR #Pers.Par.UnloadAllLeft);
END_REGION

REGION Network 29: Move piece to left
   RUNG wire#powerrail
      "PTrk_Presence"(Item := "PTrk".A0202.P["PTRK_A0202_P0"])
      Contact( #Sts.ActTargetPathLeft )
      wire#w1
      Coil( #Ctrl.Cycle.ReqMovePieceToLeft )
      I_Contact( #Sts.TrkExitLeftFull )
      I_Contact( #CIn.StopCheckQuality )
      wire#w2
      Contact( #AreaInterface.Cycle )
      wire#w3
      Coil( #Ctrl.Cycle.ExeMovePieceToLeft )
   END_RUNG
   RUNG wire#powerrail
      "PTrk_Presence"(Item := "PTrk".A0202.P["PTRK_A0202_DEVITATOR_To_EXIT"])
   END_RUNG wire#w1
   RUNG wire#w2
      Contact( #Sts.Semiautomatic )
   END_RUNG wire#w3
   // the same network as SCL:
   "PTrk_Presence"(Item := "PTrk".A0202.P["PTRK_A0202_P0"], ENO => #_w1);
   "PTrk_Presence"(Item := "PTrk".A0202.P["PTRK_A0202_DEVITATOR_To_EXIT"], ENO => #_w2);
   #Ctrl.Cycle.ReqMovePieceToLeft := (#_w1 AND #Sts.ActTargetPathLeft) OR #_w2;
   #Ctrl.Cycle.ExeMovePieceToLeft := #Ctrl.Cycle.ReqMovePieceToLeft AND NOT #Sts.TrkExitLeftFull AND NOT #CIn.StopCheckQuality AND (#AreaInterface.Cycle OR #Sts.Semiautomatic);
END_REGION

REGION Network 30: Move piece to Right
   RUNG wire#powerrail
      "PTrk_Presence"(Item := "PTrk".A0202.P["PTRK_A0202_P0"])
      Contact( #Sts.ActTargetPathRight )
      wire#w1
      Coil( #Ctrl.Cycle.ReqMovePieceToRight )
      Contact( #CIn.A03_CanLoadPiece )
      I_Contact( #CIn.StopCheckQuality )
      wire#w2
      Contact( #AreaInterface.Cycle )
      wire#w3
      Coil( #Ctrl.Cycle.ExeMovePieceToRight )
   END_RUNG
   RUNG wire#powerrail
      "PTrk_Presence"(Item := "PTrk".A0202.P["PTRK_A0202_DEVIATOR_To_A0301"])
   END_RUNG wire#w1
   RUNG wire#w2
      Contact( #Sts.Semiautomatic )
   END_RUNG wire#w3
   // the same network as SCL:
   "PTrk_Presence"(Item := "PTrk".A0202.P["PTRK_A0202_P0"], ENO => #_w1);
   "PTrk_Presence"(Item := "PTrk".A0202.P["PTRK_A0202_DEVIATOR_To_A0301"], ENO => #_w2);
   #Ctrl.Cycle.ReqMovePieceToRight := (#_w1 AND #Sts.ActTargetPathRight) OR #_w2;
   #Ctrl.Cycle.ExeMovePieceToRight := #Ctrl.Cycle.ReqMovePieceToRight AND #CIn.A03_CanLoadPiece AND NOT #CIn.StopCheckQuality AND (#AreaInterface.Cycle OR #Sts.Semiautomatic);
END_REGION

REGION Network 31: Prepare next move to left / right
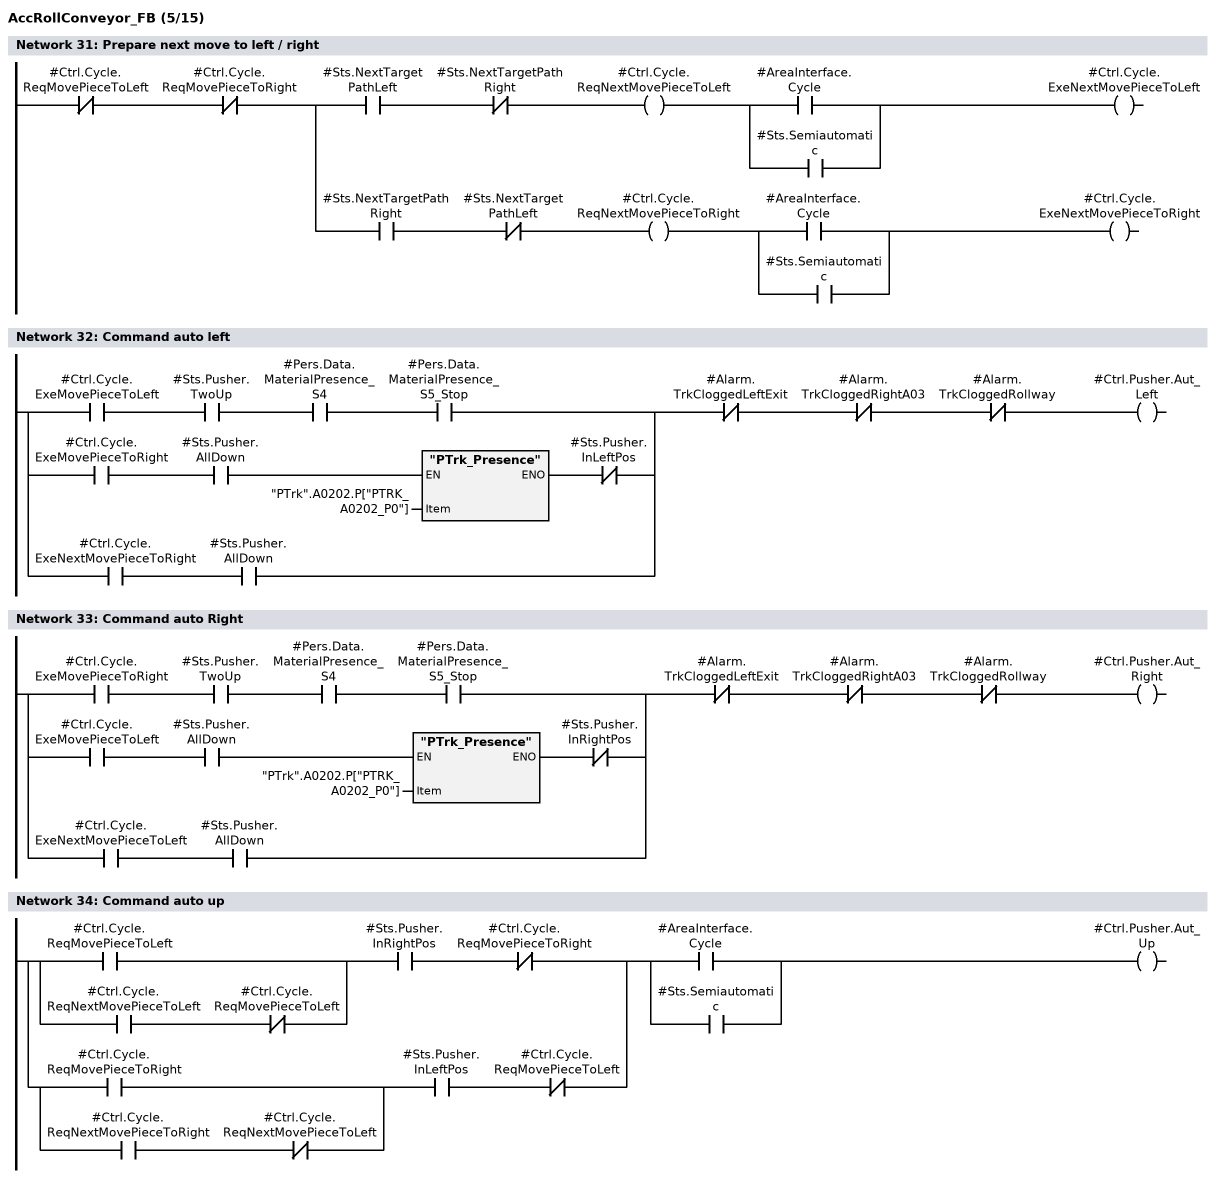
   RUNG wire#powerrail
      I_Contact( #Ctrl.Cycle.ReqMovePieceToLeft )
      I_Contact( #Ctrl.Cycle.ReqMovePieceToRight )
      wire#w1
      Contact( #Sts.NextTargetPathLeft )
      I_Contact( #Sts.NextTargetPathRight )
      Coil( #Ctrl.Cycle.ReqNextMovePieceToLeft )
      wire#w2
      Contact( #AreaInterface.Cycle )
      wire#w3
      Coil( #Ctrl.Cycle.ExeNextMovePieceToLeft )
   END_RUNG
   RUNG wire#w2
      Contact( #Sts.Semiautomatic )
   END_RUNG wire#w3
   RUNG wire#w1
      Contact( #Sts.NextTargetPathRight )
      I_Contact( #Sts.NextTargetPathLeft )
      Coil( #Ctrl.Cycle.ReqNextMovePieceToRight )
      wire#w4
      Contact( #AreaInterface.Cycle )
      wire#w5
      Coil( #Ctrl.Cycle.ExeNextMovePieceToRight )
   END_RUNG
   RUNG wire#w4
      Contact( #Sts.Semiautomatic )
   END_RUNG wire#w5
   // the same network as SCL:
   #_w1 := NOT #Ctrl.Cycle.ReqMovePieceToLeft AND NOT #Ctrl.Cycle.ReqMovePieceToRight;
   #Ctrl.Cycle.ReqNextMovePieceToLeft := #_w1 AND #Sts.NextTargetPathLeft AND NOT #Sts.NextTargetPathRight;
   #Ctrl.Cycle.ExeNextMovePieceToLeft := #Ctrl.Cycle.ReqNextMovePieceToLeft AND (#AreaInterface.Cycle OR #Sts.Semiautomatic);
   #Ctrl.Cycle.ReqNextMovePieceToRight := #_w1 AND #Sts.NextTargetPathRight AND NOT #Sts.NextTargetPathLeft;
   #Ctrl.Cycle.ExeNextMovePieceToRight := #Ctrl.Cycle.ReqNextMovePieceToRight AND (#AreaInterface.Cycle OR #Sts.Semiautomatic);
END_REGION

REGION Network 32: Command auto left
   RUNG wire#powerrail
      Contact( #Ctrl.Cycle.ExeMovePieceToLeft )
      Contact( #Sts.Pusher.TwoUp )
      Contact( #Pers.Data.MaterialPresence_S4 )
      Contact( #Pers.Data.MaterialPresence_S5_Stop )
      wire#w1
      I_Contact( #Alarm.TrkCloggedLeftExit )
      I_Contact( #Alarm.TrkCloggedRightA03 )
      I_Contact( #Alarm.TrkCloggedRollway )
      Coil( #Ctrl.Pusher.Aut_Left )
   END_RUNG
   RUNG wire#powerrail
      Contact( #Ctrl.Cycle.ExeMovePieceToRight )
      Contact( #Sts.Pusher.AllDown )
      "PTrk_Presence"(Item := "PTrk".A0202.P["PTRK_A0202_P0"])
      I_Contact( #Sts.Pusher.InLeftPos )
   END_RUNG wire#w1
   RUNG wire#powerrail
      Contact( #Ctrl.Cycle.ExeNextMovePieceToRight )
      Contact( #Sts.Pusher.AllDown )
   END_RUNG wire#w1
   // the same network as SCL:
   "PTrk_Presence"(EN := #Ctrl.Cycle.ExeMovePieceToRight AND #Sts.Pusher.AllDown,
                   Item := "PTrk".A0202.P["PTRK_A0202_P0"],
                   ENO => #_w1);
   #Ctrl.Pusher.Aut_Left := ((#Ctrl.Cycle.ExeMovePieceToLeft AND #Sts.Pusher.TwoUp AND #Pers.Data.MaterialPresence_S4 AND #Pers.Data.MaterialPresence_S5_Stop) OR (#_w1 AND NOT #Sts.Pusher.InLeftPos) OR (#Ctrl.Cycle.ExeNextMovePieceToRight AND #Sts.Pusher.AllDown)) AND NOT #Alarm.TrkCloggedLeftExit AND NOT #Alarm.TrkCloggedRightA03 AND NOT #Alarm.TrkCloggedRollway;
END_REGION

REGION Network 33: Command auto Right
   RUNG wire#powerrail
      Contact( #Ctrl.Cycle.ExeMovePieceToRight )
      Contact( #Sts.Pusher.TwoUp )
      Contact( #Pers.Data.MaterialPresence_S4 )
      Contact( #Pers.Data.MaterialPresence_S5_Stop )
      wire#w1
      I_Contact( #Alarm.TrkCloggedLeftExit )
      I_Contact( #Alarm.TrkCloggedRightA03 )
      I_Contact( #Alarm.TrkCloggedRollway )
      Coil( #Ctrl.Pusher.Aut_Right )
   END_RUNG
   RUNG wire#powerrail
      Contact( #Ctrl.Cycle.ExeMovePieceToLeft )
      Contact( #Sts.Pusher.AllDown )
      "PTrk_Presence"(Item := "PTrk".A0202.P["PTRK_A0202_P0"])
      I_Contact( #Sts.Pusher.InRightPos )
   END_RUNG wire#w1
   RUNG wire#powerrail
      Contact( #Ctrl.Cycle.ExeNextMovePieceToLeft )
      Contact( #Sts.Pusher.AllDown )
   END_RUNG wire#w1
   // the same network as SCL:
   "PTrk_Presence"(EN := #Ctrl.Cycle.ExeMovePieceToLeft AND #Sts.Pusher.AllDown,
                   Item := "PTrk".A0202.P["PTRK_A0202_P0"],
                   ENO => #_w1);
   #Ctrl.Pusher.Aut_Right := ((#Ctrl.Cycle.ExeMovePieceToRight AND #Sts.Pusher.TwoUp AND #Pers.Data.MaterialPresence_S4 AND #Pers.Data.MaterialPresence_S5_Stop) OR (#_w1 AND NOT #Sts.Pusher.InRightPos) OR (#Ctrl.Cycle.ExeNextMovePieceToLeft AND #Sts.Pusher.AllDown)) AND NOT #Alarm.TrkCloggedLeftExit AND NOT #Alarm.TrkCloggedRightA03 AND NOT #Alarm.TrkCloggedRollway;
END_REGION

REGION Network 34: Command auto up
   RUNG wire#powerrail
      Contact( #Ctrl.Cycle.ReqMovePieceToLeft )
      wire#w1
      Contact( #Sts.Pusher.InRightPos )
      I_Contact( #Ctrl.Cycle.ReqMovePieceToRight )
      wire#w2
      Contact( #AreaInterface.Cycle )
      wire#w4
      Coil( #Ctrl.Pusher.Aut_Up )
   END_RUNG
   RUNG wire#powerrail
      Contact( #Ctrl.Cycle.ReqNextMovePieceToLeft )
      I_Contact( #Ctrl.Cycle.ReqMovePieceToLeft )
   END_RUNG wire#w1
   RUNG wire#powerrail
      Contact( #Ctrl.Cycle.ReqMovePieceToRight )
      wire#w3
      Contact( #Sts.Pusher.InLeftPos )
      I_Contact( #Ctrl.Cycle.ReqMovePieceToLeft )
   END_RUNG wire#w2
   RUNG wire#powerrail
      Contact( #Ctrl.Cycle.ReqNextMovePieceToRight )
      I_Contact( #Ctrl.Cycle.ReqNextMovePieceToLeft )
   END_RUNG wire#w3
   RUNG wire#w2
      Contact( #Sts.Semiautomatic )
   END_RUNG wire#w4
   // the same network as SCL:
   #Ctrl.Pusher.Aut_Up := (((#Ctrl.Cycle.ReqMovePieceToLeft OR (#Ctrl.Cycle.ReqNextMovePieceToLeft AND NOT #Ctrl.Cycle.ReqMovePieceToLeft)) AND #Sts.Pusher.InRightPos AND NOT #Ctrl.Cycle.ReqMovePieceToRight) OR ((#Ctrl.Cycle.ReqMovePieceToRight OR (#Ctrl.Cycle.ReqNextMovePieceToRight AND NOT #Ctrl.Cycle.ReqNextMovePieceToLeft)) AND #Sts.Pusher.InLeftPos AND NOT #Ctrl.Cycle.ReqMovePieceToLeft)) AND (#AreaInterface.Cycle OR #Sts.Semiautomatic);
END_REGION

REGION Network 35: Command atuto down
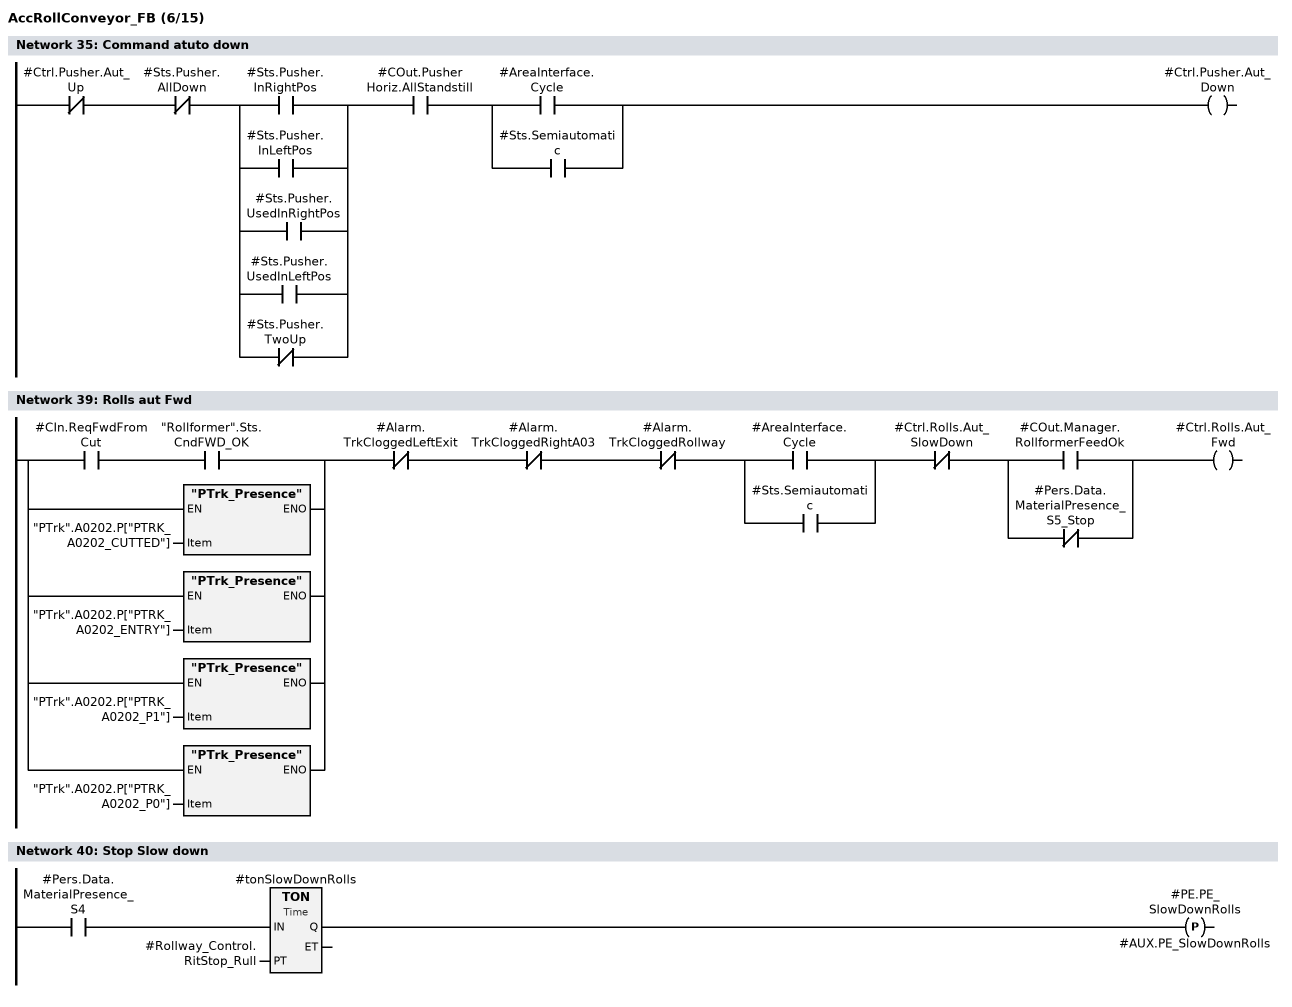
   RUNG wire#powerrail
      I_Contact( #Ctrl.Pusher.Aut_Up )
      I_Contact( #Sts.Pusher.AllDown )
      wire#w1
      Contact( #Sts.Pusher.InRightPos )
      wire#w2
      Contact( #COut.PusherHoriz.AllStandstill )
      wire#w3
      Contact( #AreaInterface.Cycle )
      wire#w4
      Coil( #Ctrl.Pusher.Aut_Down )
   END_RUNG
   RUNG wire#w1
      Contact( #Sts.Pusher.InLeftPos )
   END_RUNG wire#w2
   RUNG wire#w1
      Contact( #Sts.Pusher.UsedInRightPos )
   END_RUNG wire#w2
   RUNG wire#w1
      Contact( #Sts.Pusher.UsedInLeftPos )
   END_RUNG wire#w2
   RUNG wire#w1
      I_Contact( #Sts.Pusher.TwoUp )
   END_RUNG wire#w2
   RUNG wire#w3
      Contact( #Sts.Semiautomatic )
   END_RUNG wire#w4
   // the same network as SCL:
   #Ctrl.Pusher.Aut_Down := NOT #Ctrl.Pusher.Aut_Up AND NOT #Sts.Pusher.AllDown AND (#Sts.Pusher.InRightPos OR #Sts.Pusher.InLeftPos OR #Sts.Pusher.UsedInRightPos OR #Sts.Pusher.UsedInLeftPos OR NOT #Sts.Pusher.TwoUp) AND #COut.PusherHoriz.AllStandstill AND (#AreaInterface.Cycle OR #Sts.Semiautomatic);
END_REGION

REGION Network 36 (SCL): Pusher used
   #ActualPieceLenght := 0.0;


   IF #Ctrl.Cycle.ReqMovePieceToLeft OR
       #Ctrl.Cycle.ReqMovePieceToRight
   THEN
       IF "PTrk".A0202.P[PTRK_A0202_P0].P_ID <> 0 THEN
           #ActualPieceLenght := "PTrk".A0202.P[PTRK_A0202_P0].PLen_Meas;
       ELSIF "PTrk".A0202.P[PTRK_A0202_DEVITATOR_To_EXIT].P_ID <> 0 AND #Ctrl.Cycle.ReqMovePieceToLeft THEN
           #ActualPieceLenght := "PTrk".A0202.P[PTRK_A0202_DEVITATOR_To_EXIT].PLen_Meas;
       ELSIF "PTrk".A0202.P[PTRK_A0202_DEVIATOR_To_A0301].P_ID <> 0 AND #Ctrl.Cycle.ReqMovePieceToRight THEN
           #ActualPieceLenght := "PTrk".A0202.P[PTRK_A0202_DEVIATOR_To_A0301].PLen_Meas;
       END_IF;
   ELSIF
       #Ctrl.Cycle.ReqNextMovePieceToLeft OR
       #Ctrl.Cycle.ReqNextMovePieceToRight
   THEN
       #ActualPieceLenght := "PTrk".A0202.P[PTRK_A0202_P1].PLen_Meas;
   END_IF;


   FOR #i := 1 TO "MAX_PUSHER" DO

       IF #i = 1 THEN
           #Sts.Pusher.Used[#i] := #ActualPieceLenght <= #Pers.Par.Pusher_MaxLenghtUseFirst;
       ELSIF #i < "MAX_PUSHER" THEN

           #Sts.Pusher.Used[#i] :=
           ((#ActualPieceLenght - #Pers.Par.Pusher_DistanceFromStop[#i] > #Pers.Par.Pusher_DeltaLenghtForUse) AND NOT
           (#ActualPieceLenght - #Pers.Par.Pusher_DistanceFromStop[#i + 1] > #Pers.Par.Pusher_DeltaLenghtForUse)) OR
           (#i= 2 AND NOT #Sts.Pusher.Used[#i -1]) ;
       ELSE

           #Sts.Pusher.Used[#i] := (#ActualPieceLenght - #Pers.Par.Pusher_DistanceFromStop[#i]) > #Pers.Par.Pusher_DeltaLenghtForUse;

       END_IF;

   END_FOR;
END_REGION

REGION Network 37: >
END_REGION

REGION Network 38: <<<ROLLS MANAGER >>>
END_REGION

REGION Network 39: Rolls aut Fwd
   RUNG wire#powerrail
      Contact( #CIn.ReqFwdFromCut )
      Contact( "Rollformer".Sts.CndFWD_OK )
      wire#w1
      I_Contact( #Alarm.TrkCloggedLeftExit )
      I_Contact( #Alarm.TrkCloggedRightA03 )
      I_Contact( #Alarm.TrkCloggedRollway )
      wire#w2
      Contact( #AreaInterface.Cycle )
      wire#w3
      I_Contact( #Ctrl.Rolls.Aut_SlowDown )
      wire#w4
      Contact( #COut.Manager.RollformerFeedOk )
      wire#w5
      Coil( #Ctrl.Rolls.Aut_Fwd )
   END_RUNG
   RUNG wire#powerrail
      "PTrk_Presence"(Item := "PTrk".A0202.P["PTRK_A0202_CUTTED"])
   END_RUNG wire#w1
   RUNG wire#powerrail
      "PTrk_Presence"(Item := "PTrk".A0202.P["PTRK_A0202_ENTRY"])
   END_RUNG wire#w1
   RUNG wire#powerrail
      "PTrk_Presence"(Item := "PTrk".A0202.P["PTRK_A0202_P1"])
   END_RUNG wire#w1
   RUNG wire#powerrail
      "PTrk_Presence"(Item := "PTrk".A0202.P["PTRK_A0202_P0"])
   END_RUNG wire#w1
   RUNG wire#w2
      Contact( #Sts.Semiautomatic )
   END_RUNG wire#w3
   RUNG wire#w4
      I_Contact( #Pers.Data.MaterialPresence_S5_Stop )
   END_RUNG wire#w5
   // the same network as SCL:
   #_w2 := #CIn.ReqFwdFromCut AND "Rollformer".Sts.CndFWD_OK;
   "PTrk_Presence"(Item := "PTrk".A0202.P["PTRK_A0202_CUTTED"], ENO => #_w1);
   "PTrk_Presence"(Item := "PTrk".A0202.P["PTRK_A0202_ENTRY"], ENO => #_w3);
   "PTrk_Presence"(Item := "PTrk".A0202.P["PTRK_A0202_P1"], ENO => #_w4);
   "PTrk_Presence"(Item := "PTrk".A0202.P["PTRK_A0202_P0"], ENO => #_w5);
   #Ctrl.Rolls.Aut_Fwd := (#_w2 OR #_w1 OR #_w3 OR #_w4 OR #_w5) AND NOT #Alarm.TrkCloggedLeftExit AND NOT #Alarm.TrkCloggedRightA03 AND NOT #Alarm.TrkCloggedRollway AND (#AreaInterface.Cycle OR #Sts.Semiautomatic) AND NOT #Ctrl.Rolls.Aut_SlowDown AND (#COut.Manager.RollformerFeedOk OR NOT #Pers.Data.MaterialPresence_S5_Stop);
END_REGION

REGION Network 40: Stop Slow down
   #tonSlowDownRolls(IN := #Pers.Data.MaterialPresence_S4, PT := #Rollway_Control.RitStop_Rull);   // TON
   #PE.PE_SlowDownRolls := #tonSlowDownRolls.Q AND NOT #AUX.PE_SlowDownRolls;   // rising edge
   #AUX.PE_SlowDownRolls := #tonSlowDownRolls.Q;
END_REGION

REGION Network 41 (SCL): Stop Slow down Mem

   IF #PE.PE_SlowDownRolls THEN
       #Ctrl.Rolls.Aut_SlowDown := TRUE;
   ELSIF #Ctrl.Rolls.Aut_SlowDown AND
       (#Roll3.COut.Standstill OR
       #Roll3.COut.ActualVelocity < #Pers.Par.Rollway_StopSlowDownSpeed OR
       #Pers.Data.MaterialPresence_S5_Stop)
   THEN
       #Ctrl.Rolls.Aut_SlowDown := FALSE;
   END_IF;
END_REGION

REGION Network 42 (SCL): Piece length for speed calculation

   IF "RollformingMng".FeedLimit.PartLength <= 0.0
   THEN
       IF #Sts.TrkPieceInLenght > 0.0 THEN
           #PartLenght := #Sts.TrkPieceInLenght;
       ELSE
           #PartLenght := "PLEN_MIN_PPM_MAX";
       END_IF;
   ELSE
       #PartLenght := "RollformingMng".FeedLimit.PartLength;

   END_IF;
END_REGION

REGION Network 43: Rollss speed calculation
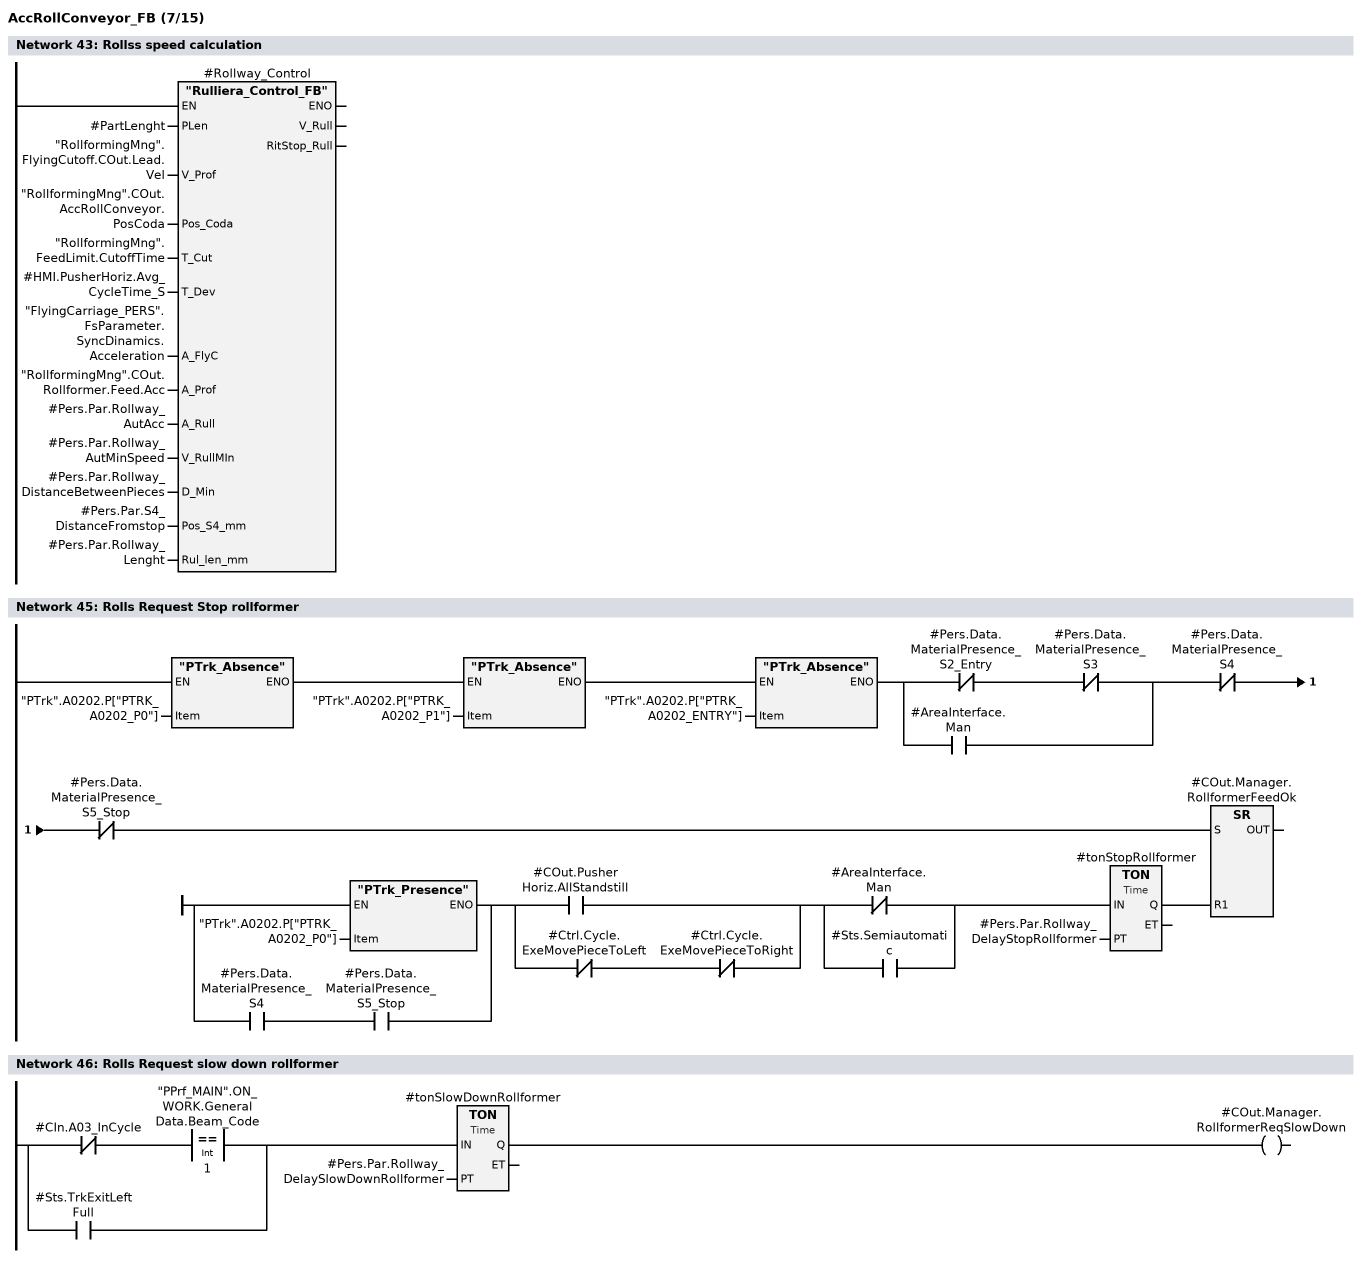
   RUNG wire#powerrail
      #Rollway_Control(PLen := #PartLenght, V_Prof := "RollformingMng".FlyingCutoff.COut.Lead.Vel, Pos_Coda := "RollformingMng".COut.AccRollConveyor.PosCoda, T_Cut := "RollformingMng".FeedLimit.CutoffTime, T_Dev := #HMI.PusherHoriz.Avg_CycleTime_S, A_FlyC := "FlyingCarriage_PERS".FsParameter.SyncDinamics.Acceleration, A_Prof := "RollformingMng".COut.Rollformer.Feed.Acc, A_Rull := #Pers.Par.Rollway_AutAcc, V_RullMIn := #Pers.Par.Rollway_AutMinSpeed, D_Min := #Pers.Par.Rollway_DistanceBetweenPieces, Pos_S4_mm := #Pers.Par.S4_DistanceFromstop, Rul_len_mm := #Pers.Par.Rollway_Lenght, V_Rull =>, RitStop_Rull =>)
   END_RUNG
   // the same network as SCL:
   #Rollway_Control(PLen := #PartLenght,   // "Rulliera_Control_FB"
                    V_Prof := "RollformingMng".FlyingCutoff.COut.Lead.Vel,
                    Pos_Coda := "RollformingMng".COut.AccRollConveyor.PosCoda,
                    T_Cut := "RollformingMng".FeedLimit.CutoffTime,
                    T_Dev := #HMI.PusherHoriz.Avg_CycleTime_S,
                    A_FlyC := "FlyingCarriage_PERS".FsParameter.SyncDinamics.Acceleration,
                    A_Prof := "RollformingMng".COut.Rollformer.Feed.Acc,
                    A_Rull := #Pers.Par.Rollway_AutAcc,
                    V_RullMIn := #Pers.Par.Rollway_AutMinSpeed,
                    D_Min := #Pers.Par.Rollway_DistanceBetweenPieces,
                    Pos_S4_mm := #Pers.Par.S4_DistanceFromstop,
                    Rul_len_mm := #Pers.Par.Rollway_Lenght);
END_REGION

REGION Network 44 (SCL): Rolls Target velocity / Acc / Dec / Jerk

   #Ctrl.Rolls.Vel := 0.0;
   #Ctrl.Rolls.Entry_Vel := 0.0;

   IF #Ctrl.Rolls.Man_Bwd OR #Ctrl.Rolls.Man_Fwd THEN

       //Prendo i dati da ultima rulliera
       #Ctrl.Rolls.Vel := #Pers.Par.Roll3.Man.VelFwdLow;
       #Ctrl.Rolls.Entry_Vel := #Pers.Par.Roll3.Man.VelFwdLow;

       #Ctrl.Rolls.Acc := #Pers.Par.Roll3.Man.Acc;
       #Ctrl.Rolls.Dec := #Pers.Par.Roll3.Man.Dec;

   ELSIF #Ctrl.Rolls.Aut_Fwd THEN


       IF #DataIn.Pb_Semiauto
       THEN
           #Ctrl.Rolls.Vel := "RollformingMng_PERS".PersistentValues.Par.SemiAut.Vel;
       ELSE


           #Ctrl.Rolls.Vel := #Rollway_Control.V_Rull;
       END_IF;

       #Ctrl.Rolls.Entry_Vel := #Ctrl.Rolls.Vel;

       #Ctrl.Rolls.Acc := #Pers.Par.Rollway_AutAcc;
       #Ctrl.Rolls.Dec := #Pers.Par.Rollway_AutDec;

   END_IF;
END_REGION

REGION Network 45: Rolls Request Stop rollformer
   RUNG wire#powerrail
      "PTrk_Absence"(Item := "PTrk".A0202.P["PTRK_A0202_P0"])
      "PTrk_Absence"(Item := "PTrk".A0202.P["PTRK_A0202_P1"])
      "PTrk_Absence"(Item := "PTrk".A0202.P["PTRK_A0202_ENTRY"])
      wire#w1
      I_Contact( #Pers.Data.MaterialPresence_S2_Entry )
      I_Contact( #Pers.Data.MaterialPresence_S3 )
      wire#w2
      I_Contact( #Pers.Data.MaterialPresence_S4 )
      I_Contact( #Pers.Data.MaterialPresence_S5_Stop )
      S_SR(operand := #COut.Manager.RollformerFeedOk, r1 := wire#w6)
   END_RUNG
   RUNG wire#w1
      Contact( #AreaInterface.Man )
   END_RUNG wire#w2
   RUNG wire#powerrail
      "PTrk_Presence"(Item := "PTrk".A0202.P["PTRK_A0202_P0"])
      wire#w3
      Contact( #COut.PusherHoriz.AllStandstill )
      wire#w4
      I_Contact( #AreaInterface.Man )
      wire#w5
      { S7_Templates := "time_type := Time" } #tonStopRollformer.TON(pt := #Pers.Par.Rollway_DelayStopRollformer, et =>)
   END_RUNG wire#w6
   RUNG wire#powerrail
      Contact( #Pers.Data.MaterialPresence_S4 )
      Contact( #Pers.Data.MaterialPresence_S5_Stop )
   END_RUNG wire#w3
   RUNG wire#w3
      I_Contact( #Ctrl.Cycle.ExeMovePieceToLeft )
      I_Contact( #Ctrl.Cycle.ExeMovePieceToRight )
   END_RUNG wire#w4
   RUNG wire#w4
      Contact( #Sts.Semiautomatic )
   END_RUNG wire#w5
   // the same network as SCL:
   "PTrk_Absence"(Item := "PTrk".A0202.P["PTRK_A0202_P0"], ENO => #_w1);
   "PTrk_Absence"(EN := #_w1, Item := "PTrk".A0202.P["PTRK_A0202_P1"], ENO => #_w2);
   "PTrk_Absence"(EN := #_w2, Item := "PTrk".A0202.P["PTRK_A0202_ENTRY"], ENO => #_w3);
   "PTrk_Presence"(Item := "PTrk".A0202.P["PTRK_A0202_P0"], ENO => #_w4);
   #tonStopRollformer(IN := (#_w4 OR (#Pers.Data.MaterialPresence_S4 AND #Pers.Data.MaterialPresence_S5_Stop)) AND (#COut.PusherHoriz.AllStandstill OR (NOT #Ctrl.Cycle.ExeMovePieceToLeft AND NOT #Ctrl.Cycle.ExeMovePieceToRight)) AND (NOT #AreaInterface.Man OR #Sts.Semiautomatic),   // TON
                      PT := #Pers.Par.Rollway_DelayStopRollformer);
   IF #_w3 AND ((NOT #Pers.Data.MaterialPresence_S2_Entry AND NOT #Pers.Data.MaterialPresence_S3) OR #AreaInterface.Man) AND NOT #Pers.Data.MaterialPresence_S4 AND NOT #Pers.Data.MaterialPresence_S5_Stop THEN
       #COut.Manager.RollformerFeedOk := TRUE;   // SR flip-flop
   END_IF;
   IF #tonStopRollformer.Q THEN #COut.Manager.RollformerFeedOk := FALSE; END_IF;
END_REGION

REGION Network 46: Rolls Request slow down rollformer
   RUNG wire#powerrail
      I_Contact( #CIn.A03_InCycle )
      { S7_Templates := "SrcType := Int" } EQ_Contact(in1 := "PPrf_MAIN".ON_WORK.GeneralData.Beam_Code, in2 := 1)
      wire#w1
      { S7_Templates := "time_type := Time" } #tonSlowDownRollformer.TON(pt := #Pers.Par.Rollway_DelaySlowDownRollformer, et =>)
      Coil( #COut.Manager.RollformerReqSlowDown )
   END_RUNG
   RUNG wire#powerrail
      Contact( #Sts.TrkExitLeftFull )
   END_RUNG wire#w1
   // the same network as SCL:
   #tonSlowDownRollformer(IN := (NOT #CIn.A03_InCycle AND ("PPrf_MAIN".ON_WORK.GeneralData.Beam_Code = 1)) OR #Sts.TrkExitLeftFull,   // TON
                          PT := #Pers.Par.Rollway_DelaySlowDownRollformer);
   #COut.Manager.RollformerReqSlowDown := #tonSlowDownRollformer.Q;
END_REGION

REGION Network 48: Comando combinato avanti/ indietro rulliere
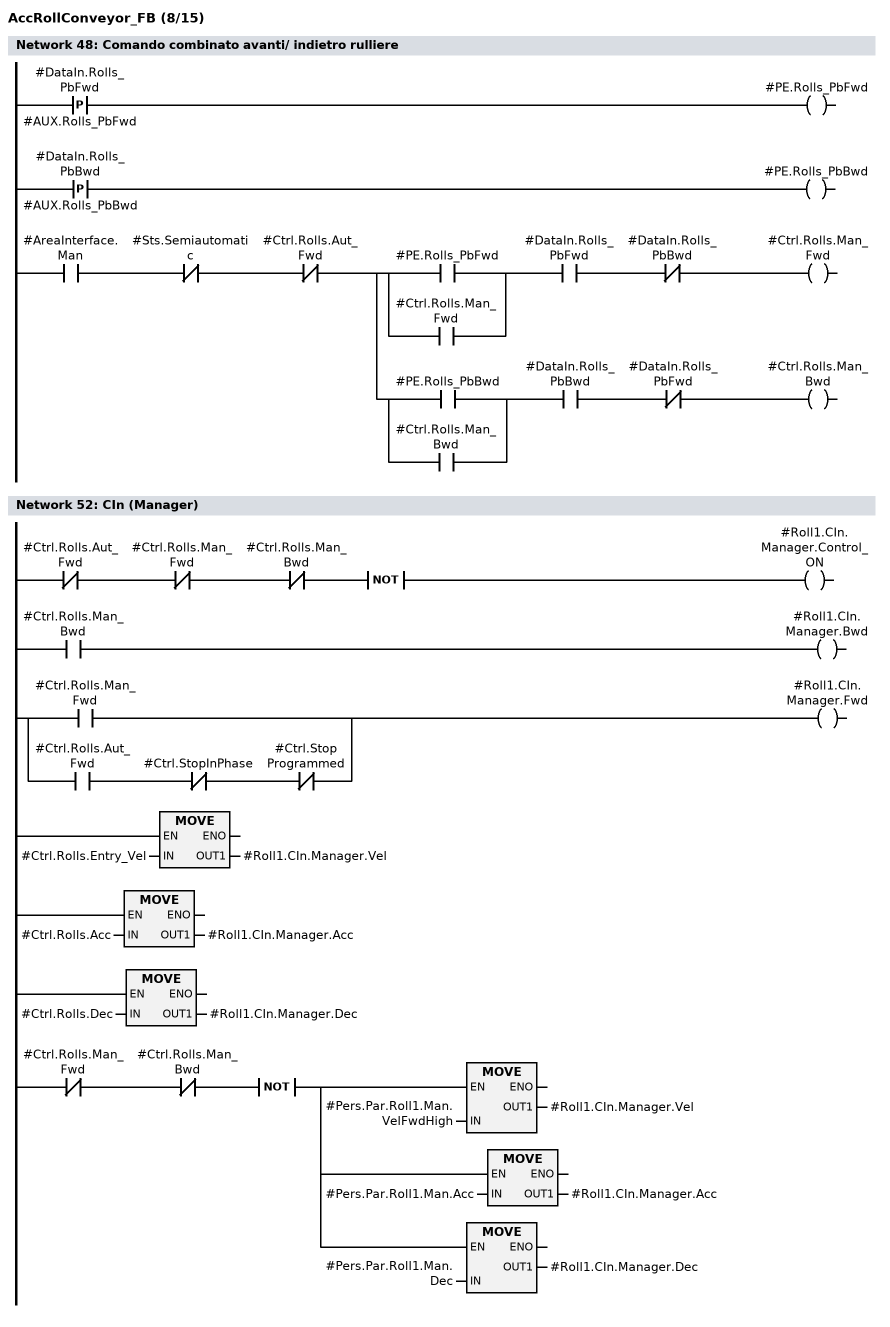
   RUNG wire#powerrail
      P_Contact(operand := #DataIn.Rolls_PbFwd, bit := #AUX.Rolls_PbFwd)
      Coil( #PE.Rolls_PbFwd )
   END_RUNG
   RUNG wire#powerrail
      P_Contact(operand := #DataIn.Rolls_PbBwd, bit := #AUX.Rolls_PbBwd)
      Coil( #PE.Rolls_PbBwd )
   END_RUNG
   RUNG wire#powerrail
      Contact( #AreaInterface.Man )
      I_Contact( #Sts.Semiautomatic )
      I_Contact( #Ctrl.Rolls.Aut_Fwd )
      wire#w1
      Contact( #PE.Rolls_PbFwd )
      wire#w2
      Contact( #DataIn.Rolls_PbFwd )
      I_Contact( #DataIn.Rolls_PbBwd )
      Coil( #Ctrl.Rolls.Man_Fwd )
   END_RUNG
   RUNG wire#w1
      Contact( #Ctrl.Rolls.Man_Fwd )
   END_RUNG wire#w2
   RUNG wire#w1
      Contact( #PE.Rolls_PbBwd )
      wire#w3
      Contact( #DataIn.Rolls_PbBwd )
      I_Contact( #DataIn.Rolls_PbFwd )
      Coil( #Ctrl.Rolls.Man_Bwd )
   END_RUNG
   RUNG wire#w1
      Contact( #Ctrl.Rolls.Man_Bwd )
   END_RUNG wire#w3
   // the same network as SCL:
   #_w1 := #DataIn.Rolls_PbFwd AND NOT #AUX.Rolls_PbFwd;   // rising edge of #DataIn.Rolls_PbFwd
   #AUX.Rolls_PbFwd := #DataIn.Rolls_PbFwd;
   #PE.Rolls_PbFwd := #_w1;
   #_w2 := #DataIn.Rolls_PbBwd AND NOT #AUX.Rolls_PbBwd;   // rising edge of #DataIn.Rolls_PbBwd
   #AUX.Rolls_PbBwd := #DataIn.Rolls_PbBwd;
   #PE.Rolls_PbBwd := #_w2;
   #_w3 := #AreaInterface.Man AND NOT #Sts.Semiautomatic AND NOT #Ctrl.Rolls.Aut_Fwd;
   #Ctrl.Rolls.Man_Fwd := #_w3 AND (#PE.Rolls_PbFwd OR #Ctrl.Rolls.Man_Fwd) AND #DataIn.Rolls_PbFwd AND NOT #DataIn.Rolls_PbBwd;
   #Ctrl.Rolls.Man_Bwd := #_w3 AND (#PE.Rolls_PbBwd OR #Ctrl.Rolls.Man_Bwd) AND #DataIn.Rolls_PbBwd AND NOT #DataIn.Rolls_PbFwd;
END_REGION

REGION Network 49: >
END_REGION

REGION Network 50: <<< ROLL 1 ENTRY >>>
END_REGION

REGION Network 51 (SCL): Cin (Manager stop)
   #Roll1.CIn.Manager.EnableStopDoorOpeningReq := #CIn.Manager.EnableStopDoorOpeningReq;
   #Roll1.CIn.Manager.EnableStopInPhase := #Ctrl.StopInPhase;
   #Roll1.CIn.Manager.EnableStopProgrammed := #Ctrl.StopProgrammed;
END_REGION

REGION Network 52: CIn (Manager)
   RUNG wire#powerrail
      I_Contact( #Ctrl.Rolls.Aut_Fwd )
      I_Contact( #Ctrl.Rolls.Man_Fwd )
      I_Contact( #Ctrl.Rolls.Man_Bwd )
      Not()
      Coil( #Roll1.CIn.Manager.Control_ON )
   END_RUNG
   RUNG wire#powerrail
      Contact( #Ctrl.Rolls.Man_Bwd )
      Coil( #Roll1.CIn.Manager.Bwd )
   END_RUNG
   RUNG wire#powerrail
      Contact( #Ctrl.Rolls.Man_Fwd )
      wire#w1
      Coil( #Roll1.CIn.Manager.Fwd )
   END_RUNG
   RUNG wire#powerrail
      Contact( #Ctrl.Rolls.Aut_Fwd )
      I_Contact( #Ctrl.StopInPhase )
      I_Contact( #Ctrl.StopProgrammed )
   END_RUNG wire#w1
   RUNG wire#powerrail
      Move(in := #Ctrl.Rolls.Entry_Vel, out1 => #Roll1.CIn.Manager.Vel)
   END_RUNG
   RUNG wire#powerrail
      Move(in := #Ctrl.Rolls.Acc, out1 => #Roll1.CIn.Manager.Acc)
   END_RUNG
   RUNG wire#powerrail
      Move(in := #Ctrl.Rolls.Dec, out1 => #Roll1.CIn.Manager.Dec)
   END_RUNG
   RUNG wire#powerrail
      I_Contact( #Ctrl.Rolls.Man_Fwd )
      I_Contact( #Ctrl.Rolls.Man_Bwd )
      Not()
      wire#w2
      Move(in := #Pers.Par.Roll1.Man.VelFwdHigh, out1 => #Roll1.CIn.Manager.Vel)
   END_RUNG
   RUNG wire#w2
      Move(in := #Pers.Par.Roll1.Man.Acc, out1 => #Roll1.CIn.Manager.Acc)
   END_RUNG
   RUNG wire#w2
      Move(in := #Pers.Par.Roll1.Man.Dec, out1 => #Roll1.CIn.Manager.Dec)
   END_RUNG
   // the same network as SCL:
   #Roll1.CIn.Manager.Control_ON := NOT (NOT #Ctrl.Rolls.Aut_Fwd AND NOT #Ctrl.Rolls.Man_Fwd AND NOT #Ctrl.Rolls.Man_Bwd);
   #Roll1.CIn.Manager.Bwd := #Ctrl.Rolls.Man_Bwd;
   #Roll1.CIn.Manager.Fwd := #Ctrl.Rolls.Man_Fwd OR (#Ctrl.Rolls.Aut_Fwd AND NOT #Ctrl.StopInPhase AND NOT #Ctrl.StopProgrammed);
   #Roll1.CIn.Manager.Vel := #Ctrl.Rolls.Entry_Vel;
   #Roll1.CIn.Manager.Acc := #Ctrl.Rolls.Acc;
   #Roll1.CIn.Manager.Dec := #Ctrl.Rolls.Dec;
   IF NOT (NOT #Ctrl.Rolls.Man_Fwd AND NOT #Ctrl.Rolls.Man_Bwd) THEN
       #Roll1.CIn.Manager.Vel := #Pers.Par.Roll1.Man.VelFwdHigh;
       #Roll1.CIn.Manager.Acc := #Pers.Par.Roll1.Man.Acc;
       #Roll1.CIn.Manager.Dec := #Pers.Par.Roll1.Man.Dec;
   END_IF;
END_REGION

REGION Network 53: CIn (External enables)
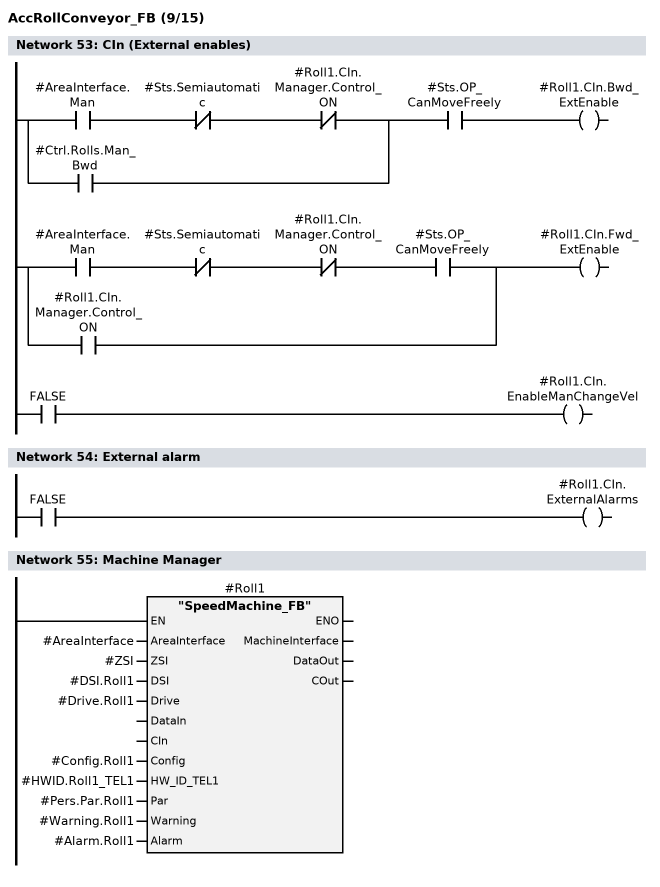
   RUNG wire#powerrail
      Contact( #AreaInterface.Man )
      I_Contact( #Sts.Semiautomatic )
      I_Contact( #Roll1.CIn.Manager.Control_ON )
      wire#w1
      Contact( #Sts.OP_CanMoveFreely )
      Coil( #Roll1.CIn.Bwd_ExtEnable )
   END_RUNG
   RUNG wire#powerrail
      Contact( #Ctrl.Rolls.Man_Bwd )
   END_RUNG wire#w1
   RUNG wire#powerrail
      Contact( #AreaInterface.Man )
      I_Contact( #Sts.Semiautomatic )
      I_Contact( #Roll1.CIn.Manager.Control_ON )
      Contact( #Sts.OP_CanMoveFreely )
      wire#w2
      Coil( #Roll1.CIn.Fwd_ExtEnable )
   END_RUNG
   RUNG wire#powerrail
      Contact( #Roll1.CIn.Manager.Control_ON )
   END_RUNG wire#w2
   RUNG wire#powerrail
      Contact( FALSE )
      Coil( #Roll1.CIn.EnableManChangeVel )
   END_RUNG
   // the same network as SCL:
   #Roll1.CIn.Bwd_ExtEnable := ((#AreaInterface.Man AND NOT #Sts.Semiautomatic AND NOT #Roll1.CIn.Manager.Control_ON) OR #Ctrl.Rolls.Man_Bwd) AND #Sts.OP_CanMoveFreely;
   #Roll1.CIn.Fwd_ExtEnable := (#AreaInterface.Man AND NOT #Sts.Semiautomatic AND NOT #Roll1.CIn.Manager.Control_ON AND #Sts.OP_CanMoveFreely) OR #Roll1.CIn.Manager.Control_ON;
   #Roll1.CIn.EnableManChangeVel := FALSE;
END_REGION

REGION Network 54: External alarm
   RUNG wire#powerrail
      Contact( FALSE )
      Coil( #Roll1.CIn.ExternalAlarms )
   END_RUNG
   // the same network as SCL:
   #Roll1.CIn.ExternalAlarms := FALSE;
END_REGION

REGION Network 55: Machine Manager
   RUNG wire#powerrail
      #Roll1(AreaInterface := #AreaInterface, ZSI := #ZSI, DSI := #DSI.Roll1, Drive := #Drive.Roll1, DataIn :=, CIn :=, Config := #Config.Roll1, HW_ID_TEL1 := #HWID.Roll1_TEL1, Par := #Pers.Par.Roll1, Warning := #Warning.Roll1, Alarm := #Alarm.Roll1, MachineInterface =>, DataOut =>, COut =>)
   END_RUNG
   // the same network as SCL:
   #Roll1(AreaInterface := #AreaInterface,   // "SpeedMachine_FB"
          ZSI := #ZSI,
          DSI := #DSI.Roll1,
          Drive := #Drive.Roll1,
          Config := #Config.Roll1,
          HW_ID_TEL1 := #HWID.Roll1_TEL1,
          Par := #Pers.Par.Roll1,
          Warning := #Warning.Roll1,
          Alarm := #Alarm.Roll1);
END_REGION

REGION Network 56: >
END_REGION

REGION Network 57: <<< ROLL 2 >>>
END_REGION

REGION Network 58 (SCL): Cin (Manager stop)
   #Roll2.CIn.Manager.EnableStopDoorOpeningReq := #CIn.Manager.EnableStopDoorOpeningReq;
   #Roll2.CIn.Manager.EnableStopInPhase := #Ctrl.StopInPhase;
   #Roll2.CIn.Manager.EnableStopProgrammed := #Ctrl.StopProgrammed;
END_REGION

REGION Network 59: CIn (Manager)
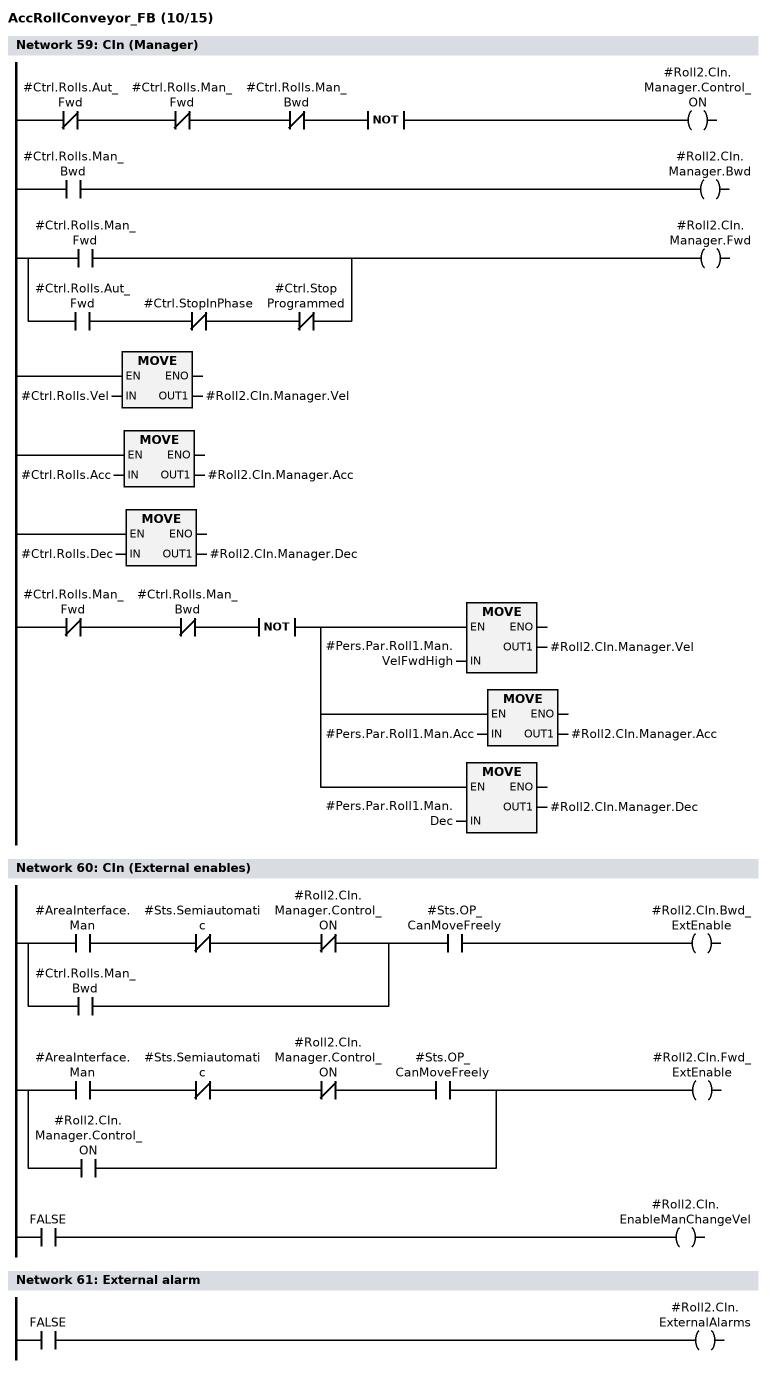
   RUNG wire#powerrail
      I_Contact( #Ctrl.Rolls.Aut_Fwd )
      I_Contact( #Ctrl.Rolls.Man_Fwd )
      I_Contact( #Ctrl.Rolls.Man_Bwd )
      Not()
      Coil( #Roll2.CIn.Manager.Control_ON )
   END_RUNG
   RUNG wire#powerrail
      Contact( #Ctrl.Rolls.Man_Bwd )
      Coil( #Roll2.CIn.Manager.Bwd )
   END_RUNG
   RUNG wire#powerrail
      Contact( #Ctrl.Rolls.Man_Fwd )
      wire#w1
      Coil( #Roll2.CIn.Manager.Fwd )
   END_RUNG
   RUNG wire#powerrail
      Contact( #Ctrl.Rolls.Aut_Fwd )
      I_Contact( #Ctrl.StopInPhase )
      I_Contact( #Ctrl.StopProgrammed )
   END_RUNG wire#w1
   RUNG wire#powerrail
      Move(in := #Ctrl.Rolls.Vel, out1 => #Roll2.CIn.Manager.Vel)
   END_RUNG
   RUNG wire#powerrail
      Move(in := #Ctrl.Rolls.Acc, out1 => #Roll2.CIn.Manager.Acc)
   END_RUNG
   RUNG wire#powerrail
      Move(in := #Ctrl.Rolls.Dec, out1 => #Roll2.CIn.Manager.Dec)
   END_RUNG
   RUNG wire#powerrail
      I_Contact( #Ctrl.Rolls.Man_Fwd )
      I_Contact( #Ctrl.Rolls.Man_Bwd )
      Not()
      wire#w2
      Move(in := #Pers.Par.Roll1.Man.VelFwdHigh, out1 => #Roll2.CIn.Manager.Vel)
   END_RUNG
   RUNG wire#w2
      Move(in := #Pers.Par.Roll1.Man.Acc, out1 => #Roll2.CIn.Manager.Acc)
   END_RUNG
   RUNG wire#w2
      Move(in := #Pers.Par.Roll1.Man.Dec, out1 => #Roll2.CIn.Manager.Dec)
   END_RUNG
   // the same network as SCL:
   #Roll2.CIn.Manager.Control_ON := NOT (NOT #Ctrl.Rolls.Aut_Fwd AND NOT #Ctrl.Rolls.Man_Fwd AND NOT #Ctrl.Rolls.Man_Bwd);
   #Roll2.CIn.Manager.Bwd := #Ctrl.Rolls.Man_Bwd;
   #Roll2.CIn.Manager.Fwd := #Ctrl.Rolls.Man_Fwd OR (#Ctrl.Rolls.Aut_Fwd AND NOT #Ctrl.StopInPhase AND NOT #Ctrl.StopProgrammed);
   #Roll2.CIn.Manager.Vel := #Ctrl.Rolls.Vel;
   #Roll2.CIn.Manager.Acc := #Ctrl.Rolls.Acc;
   #Roll2.CIn.Manager.Dec := #Ctrl.Rolls.Dec;
   IF NOT (NOT #Ctrl.Rolls.Man_Fwd AND NOT #Ctrl.Rolls.Man_Bwd) THEN
       #Roll2.CIn.Manager.Vel := #Pers.Par.Roll1.Man.VelFwdHigh;
       #Roll2.CIn.Manager.Acc := #Pers.Par.Roll1.Man.Acc;
       #Roll2.CIn.Manager.Dec := #Pers.Par.Roll1.Man.Dec;
   END_IF;
END_REGION

REGION Network 60: CIn (External enables)
   RUNG wire#powerrail
      Contact( #AreaInterface.Man )
      I_Contact( #Sts.Semiautomatic )
      I_Contact( #Roll2.CIn.Manager.Control_ON )
      wire#w1
      Contact( #Sts.OP_CanMoveFreely )
      Coil( #Roll2.CIn.Bwd_ExtEnable )
   END_RUNG
   RUNG wire#powerrail
      Contact( #Ctrl.Rolls.Man_Bwd )
   END_RUNG wire#w1
   RUNG wire#powerrail
      Contact( #AreaInterface.Man )
      I_Contact( #Sts.Semiautomatic )
      I_Contact( #Roll2.CIn.Manager.Control_ON )
      Contact( #Sts.OP_CanMoveFreely )
      wire#w2
      Coil( #Roll2.CIn.Fwd_ExtEnable )
   END_RUNG
   RUNG wire#powerrail
      Contact( #Roll2.CIn.Manager.Control_ON )
   END_RUNG wire#w2
   RUNG wire#powerrail
      Contact( FALSE )
      Coil( #Roll2.CIn.EnableManChangeVel )
   END_RUNG
   // the same network as SCL:
   #Roll2.CIn.Bwd_ExtEnable := ((#AreaInterface.Man AND NOT #Sts.Semiautomatic AND NOT #Roll2.CIn.Manager.Control_ON) OR #Ctrl.Rolls.Man_Bwd) AND #Sts.OP_CanMoveFreely;
   #Roll2.CIn.Fwd_ExtEnable := (#AreaInterface.Man AND NOT #Sts.Semiautomatic AND NOT #Roll2.CIn.Manager.Control_ON AND #Sts.OP_CanMoveFreely) OR #Roll2.CIn.Manager.Control_ON;
   #Roll2.CIn.EnableManChangeVel := FALSE;
END_REGION

REGION Network 61: External alarm
   RUNG wire#powerrail
      Contact( FALSE )
      Coil( #Roll2.CIn.ExternalAlarms )
   END_RUNG
   // the same network as SCL:
   #Roll2.CIn.ExternalAlarms := FALSE;
END_REGION

REGION Network 62: Machine Manager
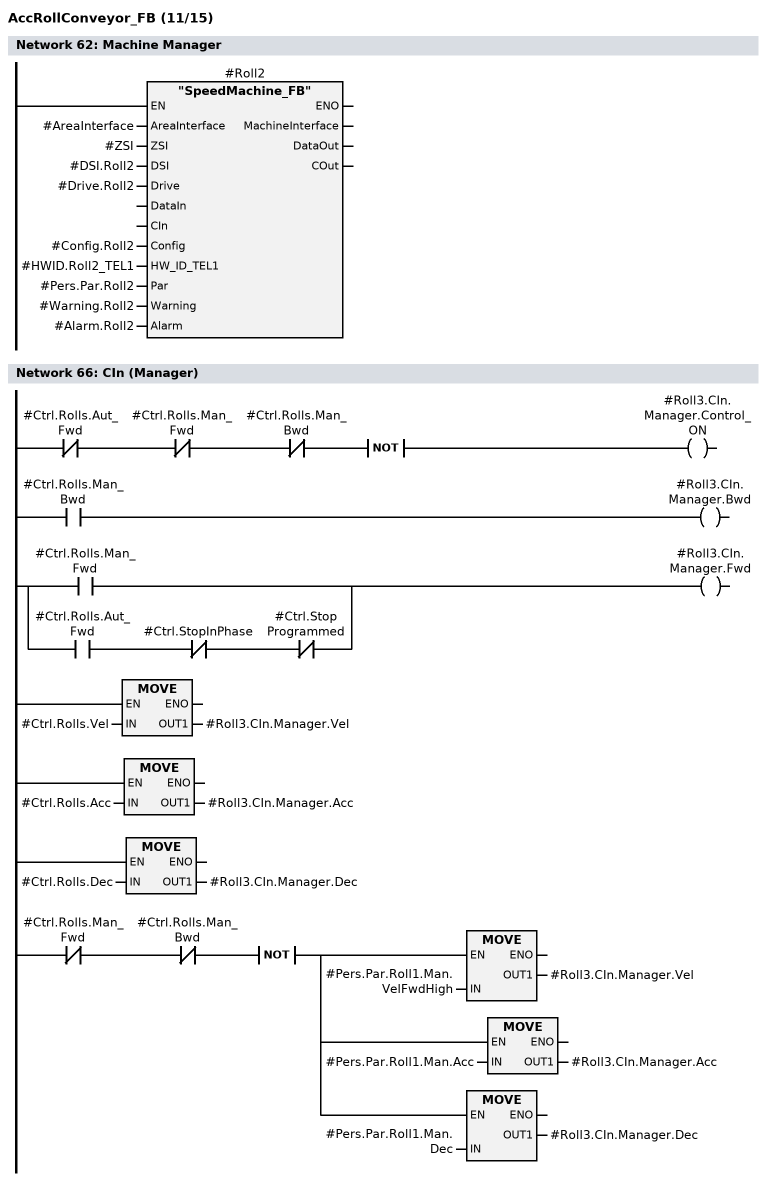
   RUNG wire#powerrail
      #Roll2(AreaInterface := #AreaInterface, ZSI := #ZSI, DSI := #DSI.Roll2, Drive := #Drive.Roll2, DataIn :=, CIn :=, Config := #Config.Roll2, HW_ID_TEL1 := #HWID.Roll2_TEL1, Par := #Pers.Par.Roll2, Warning := #Warning.Roll2, Alarm := #Alarm.Roll2, MachineInterface =>, DataOut =>, COut =>)
   END_RUNG
   // the same network as SCL:
   #Roll2(AreaInterface := #AreaInterface,   // "SpeedMachine_FB"
          ZSI := #ZSI,
          DSI := #DSI.Roll2,
          Drive := #Drive.Roll2,
          Config := #Config.Roll2,
          HW_ID_TEL1 := #HWID.Roll2_TEL1,
          Par := #Pers.Par.Roll2,
          Warning := #Warning.Roll2,
          Alarm := #Alarm.Roll2);
END_REGION

REGION Network 63: >
END_REGION

REGION Network 64: <<< ROLL 3 >>>
END_REGION

REGION Network 65 (SCL): Cin (Manager stop)
   #Roll3.CIn.Manager.EnableStopDoorOpeningReq := #CIn.Manager.EnableStopDoorOpeningReq;
   #Roll3.CIn.Manager.EnableStopInPhase := #Ctrl.StopInPhase;
   #Roll3.CIn.Manager.EnableStopProgrammed := #Ctrl.StopProgrammed;
END_REGION

REGION Network 66: CIn (Manager)
   RUNG wire#powerrail
      I_Contact( #Ctrl.Rolls.Aut_Fwd )
      I_Contact( #Ctrl.Rolls.Man_Fwd )
      I_Contact( #Ctrl.Rolls.Man_Bwd )
      Not()
      Coil( #Roll3.CIn.Manager.Control_ON )
   END_RUNG
   RUNG wire#powerrail
      Contact( #Ctrl.Rolls.Man_Bwd )
      Coil( #Roll3.CIn.Manager.Bwd )
   END_RUNG
   RUNG wire#powerrail
      Contact( #Ctrl.Rolls.Man_Fwd )
      wire#w1
      Coil( #Roll3.CIn.Manager.Fwd )
   END_RUNG
   RUNG wire#powerrail
      Contact( #Ctrl.Rolls.Aut_Fwd )
      I_Contact( #Ctrl.StopInPhase )
      I_Contact( #Ctrl.StopProgrammed )
   END_RUNG wire#w1
   RUNG wire#powerrail
      Move(in := #Ctrl.Rolls.Vel, out1 => #Roll3.CIn.Manager.Vel)
   END_RUNG
   RUNG wire#powerrail
      Move(in := #Ctrl.Rolls.Acc, out1 => #Roll3.CIn.Manager.Acc)
   END_RUNG
   RUNG wire#powerrail
      Move(in := #Ctrl.Rolls.Dec, out1 => #Roll3.CIn.Manager.Dec)
   END_RUNG
   RUNG wire#powerrail
      I_Contact( #Ctrl.Rolls.Man_Fwd )
      I_Contact( #Ctrl.Rolls.Man_Bwd )
      Not()
      wire#w2
      Move(in := #Pers.Par.Roll1.Man.VelFwdHigh, out1 => #Roll3.CIn.Manager.Vel)
   END_RUNG
   RUNG wire#w2
      Move(in := #Pers.Par.Roll1.Man.Acc, out1 => #Roll3.CIn.Manager.Acc)
   END_RUNG
   RUNG wire#w2
      Move(in := #Pers.Par.Roll1.Man.Dec, out1 => #Roll3.CIn.Manager.Dec)
   END_RUNG
   // the same network as SCL:
   #Roll3.CIn.Manager.Control_ON := NOT (NOT #Ctrl.Rolls.Aut_Fwd AND NOT #Ctrl.Rolls.Man_Fwd AND NOT #Ctrl.Rolls.Man_Bwd);
   #Roll3.CIn.Manager.Bwd := #Ctrl.Rolls.Man_Bwd;
   #Roll3.CIn.Manager.Fwd := #Ctrl.Rolls.Man_Fwd OR (#Ctrl.Rolls.Aut_Fwd AND NOT #Ctrl.StopInPhase AND NOT #Ctrl.StopProgrammed);
   #Roll3.CIn.Manager.Vel := #Ctrl.Rolls.Vel;
   #Roll3.CIn.Manager.Acc := #Ctrl.Rolls.Acc;
   #Roll3.CIn.Manager.Dec := #Ctrl.Rolls.Dec;
   IF NOT (NOT #Ctrl.Rolls.Man_Fwd AND NOT #Ctrl.Rolls.Man_Bwd) THEN
       #Roll3.CIn.Manager.Vel := #Pers.Par.Roll1.Man.VelFwdHigh;
       #Roll3.CIn.Manager.Acc := #Pers.Par.Roll1.Man.Acc;
       #Roll3.CIn.Manager.Dec := #Pers.Par.Roll1.Man.Dec;
   END_IF;
END_REGION

REGION Network 67: CIn (External enables)
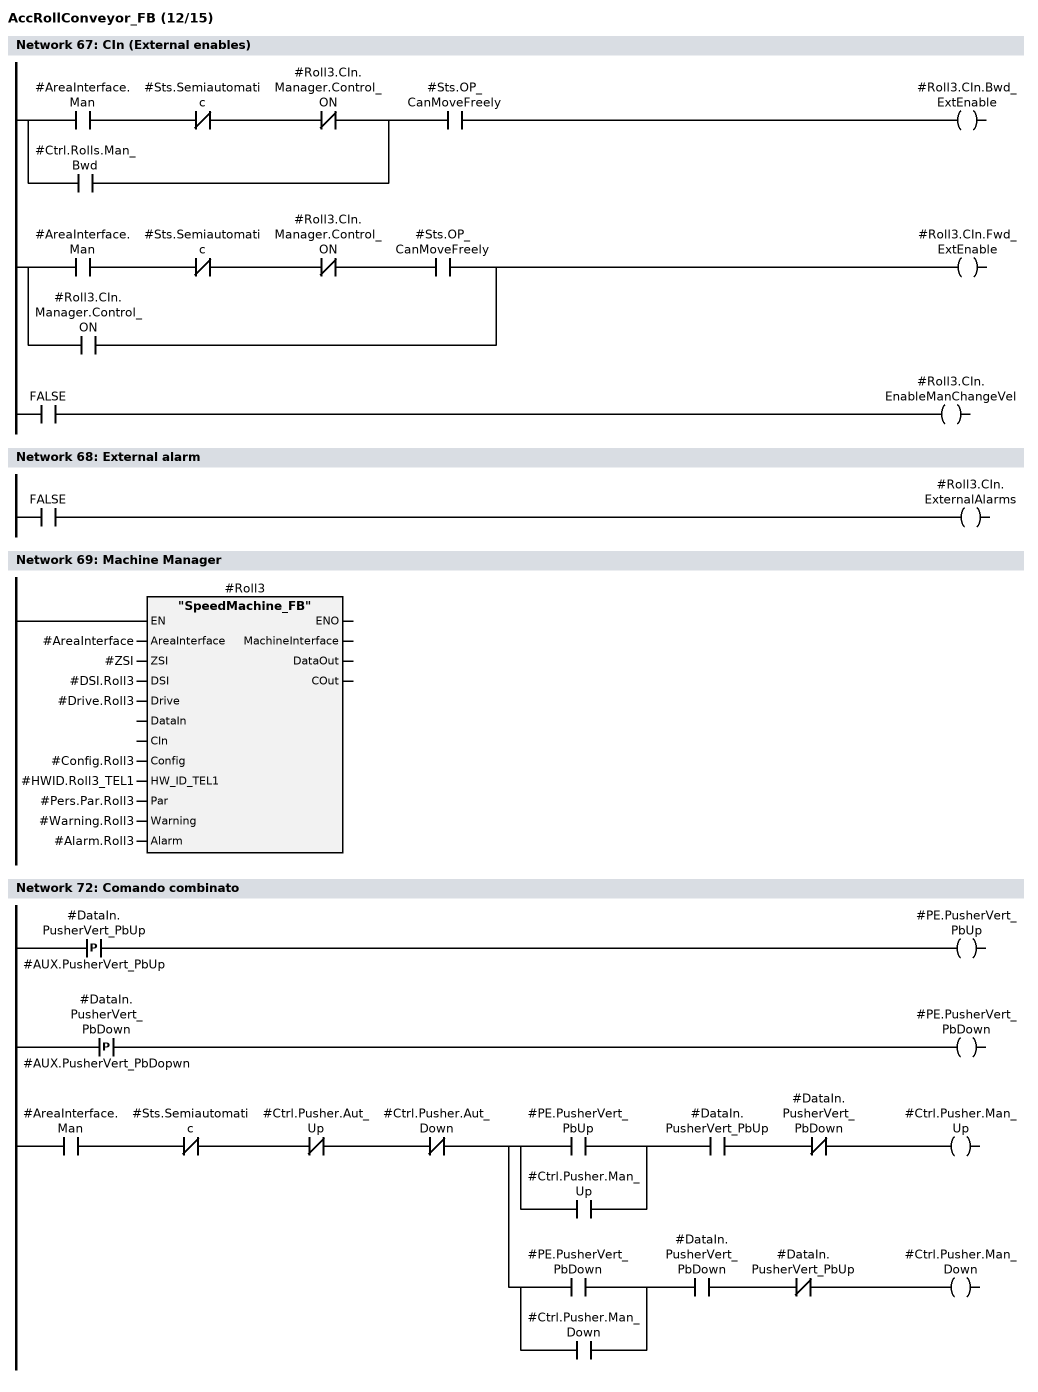
   RUNG wire#powerrail
      Contact( #AreaInterface.Man )
      I_Contact( #Sts.Semiautomatic )
      I_Contact( #Roll3.CIn.Manager.Control_ON )
      wire#w1
      Contact( #Sts.OP_CanMoveFreely )
      Coil( #Roll3.CIn.Bwd_ExtEnable )
   END_RUNG
   RUNG wire#powerrail
      Contact( #Ctrl.Rolls.Man_Bwd )
   END_RUNG wire#w1
   RUNG wire#powerrail
      Contact( #AreaInterface.Man )
      I_Contact( #Sts.Semiautomatic )
      I_Contact( #Roll3.CIn.Manager.Control_ON )
      Contact( #Sts.OP_CanMoveFreely )
      wire#w2
      Coil( #Roll3.CIn.Fwd_ExtEnable )
   END_RUNG
   RUNG wire#powerrail
      Contact( #Roll3.CIn.Manager.Control_ON )
   END_RUNG wire#w2
   RUNG wire#powerrail
      Contact( FALSE )
      Coil( #Roll3.CIn.EnableManChangeVel )
   END_RUNG
   // the same network as SCL:
   #Roll3.CIn.Bwd_ExtEnable := ((#AreaInterface.Man AND NOT #Sts.Semiautomatic AND NOT #Roll3.CIn.Manager.Control_ON) OR #Ctrl.Rolls.Man_Bwd) AND #Sts.OP_CanMoveFreely;
   #Roll3.CIn.Fwd_ExtEnable := (#AreaInterface.Man AND NOT #Sts.Semiautomatic AND NOT #Roll3.CIn.Manager.Control_ON AND #Sts.OP_CanMoveFreely) OR #Roll3.CIn.Manager.Control_ON;
   #Roll3.CIn.EnableManChangeVel := FALSE;
END_REGION

REGION Network 68: External alarm
   RUNG wire#powerrail
      Contact( FALSE )
      Coil( #Roll3.CIn.ExternalAlarms )
   END_RUNG
   // the same network as SCL:
   #Roll3.CIn.ExternalAlarms := FALSE;
END_REGION

REGION Network 69: Machine Manager
   RUNG wire#powerrail
      #Roll3(AreaInterface := #AreaInterface, ZSI := #ZSI, DSI := #DSI.Roll3, Drive := #Drive.Roll3, DataIn :=, CIn :=, Config := #Config.Roll3, HW_ID_TEL1 := #HWID.Roll3_TEL1, Par := #Pers.Par.Roll3, Warning := #Warning.Roll3, Alarm := #Alarm.Roll3, MachineInterface =>, DataOut =>, COut =>)
   END_RUNG
   // the same network as SCL:
   #Roll3(AreaInterface := #AreaInterface,   // "SpeedMachine_FB"
          ZSI := #ZSI,
          DSI := #DSI.Roll3,
          Drive := #Drive.Roll3,
          Config := #Config.Roll3,
          HW_ID_TEL1 := #HWID.Roll3_TEL1,
          Par := #Pers.Par.Roll3,
          Warning := #Warning.Roll3,
          Alarm := #Alarm.Roll3);
END_REGION

REGION Network 70: >
END_REGION

REGION Network 71: <<< PUSHER VERT >>>
END_REGION

REGION Network 72: Comando combinato
   RUNG wire#powerrail
      P_Contact(operand := #DataIn.PusherVert_PbUp, bit := #AUX.PusherVert_PbUp)
      Coil( #PE.PusherVert_PbUp )
   END_RUNG
   RUNG wire#powerrail
      P_Contact(operand := #DataIn.PusherVert_PbDown, bit := #AUX.PusherVert_PbDopwn)
      Coil( #PE.PusherVert_PbDown )
   END_RUNG
   RUNG wire#powerrail
      Contact( #AreaInterface.Man )
      I_Contact( #Sts.Semiautomatic )
      I_Contact( #Ctrl.Pusher.Aut_Up )
      I_Contact( #Ctrl.Pusher.Aut_Down )
      wire#w1
      Contact( #PE.PusherVert_PbUp )
      wire#w2
      Contact( #DataIn.PusherVert_PbUp )
      I_Contact( #DataIn.PusherVert_PbDown )
      Coil( #Ctrl.Pusher.Man_Up )
   END_RUNG
   RUNG wire#w1
      Contact( #Ctrl.Pusher.Man_Up )
   END_RUNG wire#w2
   RUNG wire#w1
      Contact( #PE.PusherVert_PbDown )
      wire#w3
      Contact( #DataIn.PusherVert_PbDown )
      I_Contact( #DataIn.PusherVert_PbUp )
      Coil( #Ctrl.Pusher.Man_Down )
   END_RUNG
   RUNG wire#w1
      Contact( #Ctrl.Pusher.Man_Down )
   END_RUNG wire#w3
   // the same network as SCL:
   #_w1 := #DataIn.PusherVert_PbUp AND NOT #AUX.PusherVert_PbUp;   // rising edge of #DataIn.PusherVert_PbUp
   #AUX.PusherVert_PbUp := #DataIn.PusherVert_PbUp;
   #PE.PusherVert_PbUp := #_w1;
   #_w2 := #DataIn.PusherVert_PbDown AND NOT #AUX.PusherVert_PbDopwn;   // rising edge of #DataIn.PusherVert_PbDown
   #AUX.PusherVert_PbDopwn := #DataIn.PusherVert_PbDown;
   #PE.PusherVert_PbDown := #_w2;
   #_w3 := #AreaInterface.Man AND NOT #Sts.Semiautomatic AND NOT #Ctrl.Pusher.Aut_Up AND NOT #Ctrl.Pusher.Aut_Down;
   #Ctrl.Pusher.Man_Up := #_w3 AND (#PE.PusherVert_PbUp OR #Ctrl.Pusher.Man_Up) AND #DataIn.PusherVert_PbUp AND NOT #DataIn.PusherVert_PbDown;
   #Ctrl.Pusher.Man_Down := #_w3 AND (#PE.PusherVert_PbDown OR #Ctrl.Pusher.Man_Down) AND #DataIn.PusherVert_PbDown AND NOT #DataIn.PusherVert_PbUp;
END_REGION

REGION Network 73 (SCL): Manager

   #PusherVert_MachineInterface := #PusherVert[1].MachineInterface;
   #Sts.Pusher.AllDown := TRUE;
   #PusherVert_NrUp := 0;

   #COut.PusherVert.AllStandstill := TRUE;
   #COut.PusherVert.Rest_CheckNext := FALSE;
   #COut.PusherVert.Work_CheckNext := FALSE;

   FOR #i := 1 TO "MAX_PUSHER" DO

       #PusherVert[#i].Cin.Manager.EnableStopDoorOpeningReq := #CIn.Manager.EnableStopDoorOpeningReq;
       #PusherVert[#i].Cin.Manager.EnableStopInPhase := #Ctrl.StopInPhase;
       #PusherVert[#i].Cin.Manager.EnableStopProgrammed := #Ctrl.StopProgrammed;

       #PusherVert[#i].Cin.Manager.Control_ON := #Ctrl.Pusher.Aut_Down OR #Ctrl.Pusher.Aut_Up OR #Ctrl.Pusher.Man_Down OR #Ctrl.Pusher.Man_Up;
       #PusherVert[#i].Cin.Manager.Work := (#Ctrl.Pusher.Aut_Up AND #Sts.Pusher.Used[#i] AND NOT #Ctrl.StopInPhase AND NOT #Ctrl.StopProgrammed) OR #Ctrl.Pusher.Man_Up;
       #PusherVert[#i].Cin.Manager.Rest := (#Ctrl.Pusher.Aut_Down AND NOT #Ctrl.StopInPhase AND NOT #Ctrl.StopProgrammed) OR #Ctrl.Pusher.Man_Down;

       #PusherVert[#i].Cin.Rest_ExtEnable := TRUE;
       #PusherVert[#i].Cin.Work_ExtEnable := (#AreaInterface.Man AND NOT #Sts.Semiautomatic AND #Sts.OP_CanMoveFreely) OR (#PusherVert[#i].Cin.Manager.Control_ON AND #Sts.Pusher.Used[#i]);
       #PusherVert[#i].Cin.ExternalAlarms := FALSE;


       #PusherVert[#i](AreaInterface := #AreaInterface,
                       ZSI := #ZSI,
                       DSI := #DSI.PusherVert,
                       Config := #Config.PusherVert[#i],
                       Alarm := #Alarm.PusherVert[#i],
                       Warning := #Warning.PusherVert[#i]);


       IF NOT #PusherVert[#i].COut.Rest THEN
           #Sts.Pusher.AllDown := FALSE;
       END_IF;
       IF #PusherVert[#i].COut.Work THEN
           #PusherVert_NrUp += 1;
       END_IF;
       IF NOT #PusherVert[#i].COut.Standstill THEN
           #COut.PusherVert.AllStandstill := FALSE;
       END_IF;
       IF #PusherVert[#i].COut.Rest_CheckNext THEN
           #COut.PusherVert.Rest_CheckNext := TRUE;
       END_IF;
       IF #PusherVert[#i].COut.Work_CheckNext THEN
           #COut.PusherVert.Work_CheckNext := TRUE;
       END_IF;


       IF #i = 1 THEN
           #PusherVert_MachineInterface := #PusherVert[#i].MachineInterface;
       ELSE
           #PusherVert_MachineInterface := "MachineInterface_2_To_1"(MachineInterface_1 := #PusherVert_MachineInterface,
                                                                      MachineInterface_2 := #PusherVert[#i].MachineInterface,
                                                                      AdditionalAlarms := FALSE,
                                                                      AdditionalWarnings := FALSE);
       END_IF;
   END_FOR;

   #Sts.Pusher.TwoUp := #PusherVert_NrUp >= 2;
   #COut.PusherVert.TwoUp := #Sts.Pusher.TwoUp;
   #COut.PusherVert.AllDown := #Sts.Pusher.AllDown;
END_REGION

REGION Network 74: >
END_REGION

REGION Network 75: <<< PUSHER HORIZ >>>
END_REGION

REGION Network 76: Comando combinato
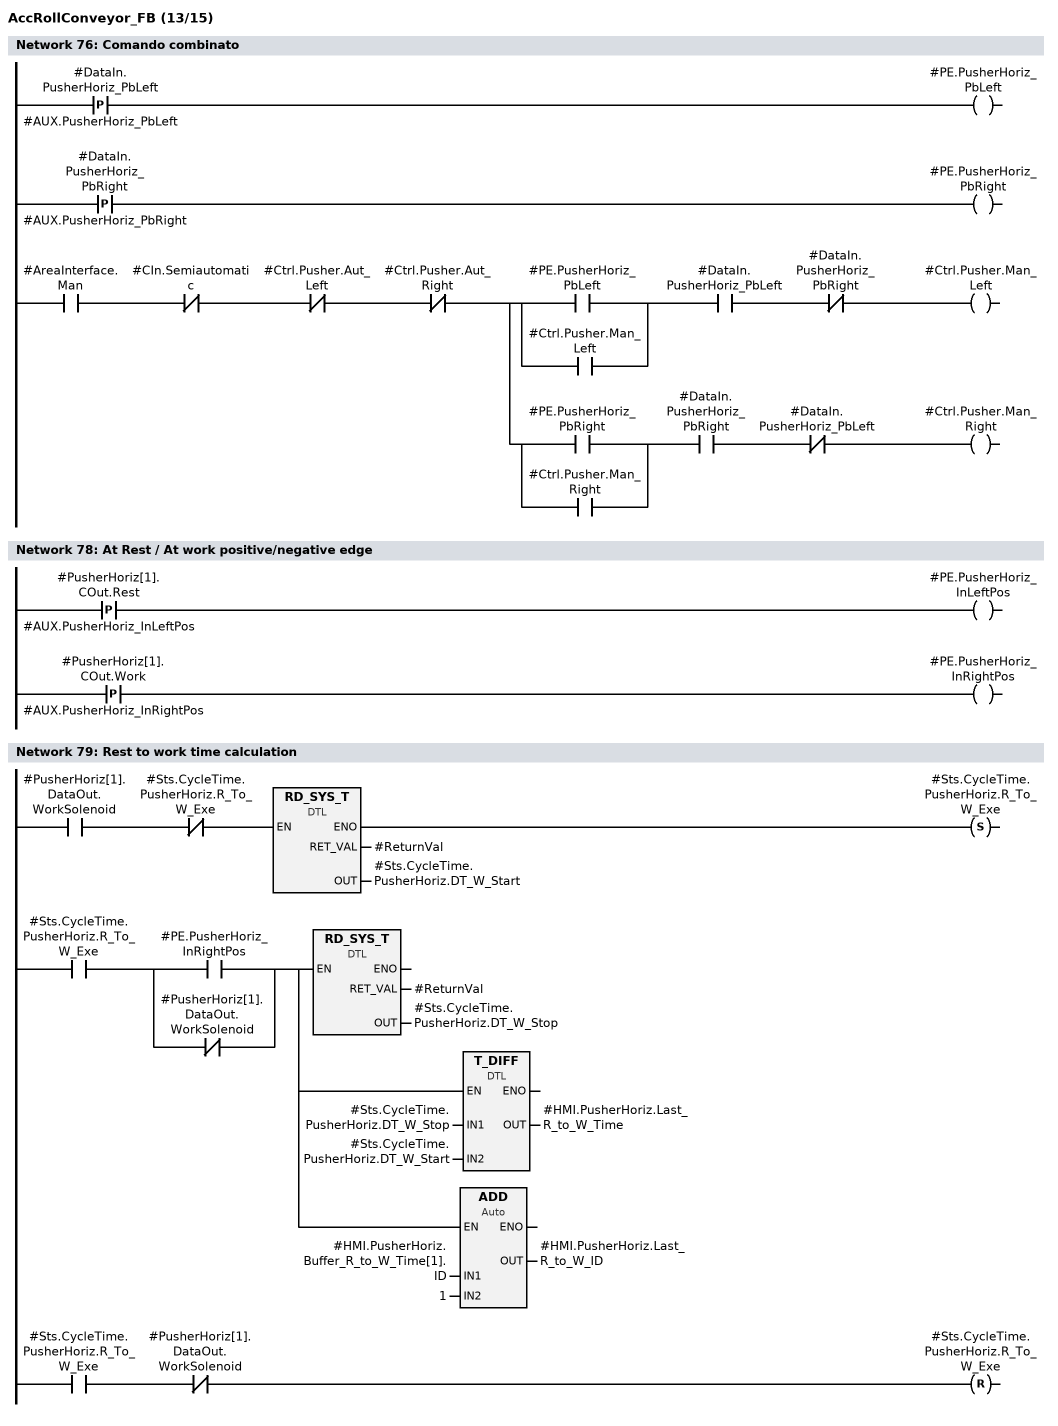
   RUNG wire#powerrail
      P_Contact(operand := #DataIn.PusherHoriz_PbLeft, bit := #AUX.PusherHoriz_PbLeft)
      Coil( #PE.PusherHoriz_PbLeft )
   END_RUNG
   RUNG wire#powerrail
      P_Contact(operand := #DataIn.PusherHoriz_PbRight, bit := #AUX.PusherHoriz_PbRight)
      Coil( #PE.PusherHoriz_PbRight )
   END_RUNG
   RUNG wire#powerrail
      Contact( #AreaInterface.Man )
      I_Contact( #CIn.Semiautomatic )
      I_Contact( #Ctrl.Pusher.Aut_Left )
      I_Contact( #Ctrl.Pusher.Aut_Right )
      wire#w1
      Contact( #PE.PusherHoriz_PbLeft )
      wire#w2
      Contact( #DataIn.PusherHoriz_PbLeft )
      I_Contact( #DataIn.PusherHoriz_PbRight )
      Coil( #Ctrl.Pusher.Man_Left )
   END_RUNG
   RUNG wire#w1
      Contact( #Ctrl.Pusher.Man_Left )
   END_RUNG wire#w2
   RUNG wire#w1
      Contact( #PE.PusherHoriz_PbRight )
      wire#w3
      Contact( #DataIn.PusherHoriz_PbRight )
      I_Contact( #DataIn.PusherHoriz_PbLeft )
      Coil( #Ctrl.Pusher.Man_Right )
   END_RUNG
   RUNG wire#w1
      Contact( #Ctrl.Pusher.Man_Right )
   END_RUNG wire#w3
   // the same network as SCL:
   #_w1 := #DataIn.PusherHoriz_PbLeft AND NOT #AUX.PusherHoriz_PbLeft;   // rising edge of #DataIn.PusherHoriz_PbLeft
   #AUX.PusherHoriz_PbLeft := #DataIn.PusherHoriz_PbLeft;
   #PE.PusherHoriz_PbLeft := #_w1;
   #_w2 := #DataIn.PusherHoriz_PbRight AND NOT #AUX.PusherHoriz_PbRight;   // rising edge of #DataIn.PusherHoriz_PbRight
   #AUX.PusherHoriz_PbRight := #DataIn.PusherHoriz_PbRight;
   #PE.PusherHoriz_PbRight := #_w2;
   #_w3 := #AreaInterface.Man AND NOT #CIn.Semiautomatic AND NOT #Ctrl.Pusher.Aut_Left AND NOT #Ctrl.Pusher.Aut_Right;
   #Ctrl.Pusher.Man_Left := #_w3 AND (#PE.PusherHoriz_PbLeft OR #Ctrl.Pusher.Man_Left) AND #DataIn.PusherHoriz_PbLeft AND NOT #DataIn.PusherHoriz_PbRight;
   #Ctrl.Pusher.Man_Right := #_w3 AND (#PE.PusherHoriz_PbRight OR #Ctrl.Pusher.Man_Right) AND #DataIn.PusherHoriz_PbRight AND NOT #DataIn.PusherHoriz_PbLeft;
END_REGION

REGION Network 77 (SCL): Manager

   #PusherHoriz_MachineInterface := #PusherHoriz[1].MachineInterface;
   #Sts.Pusher.InLeftPos  := TRUE;
   #Sts.Pusher.InRightPos := TRUE;
   #Sts.Pusher.UsedInLeftPos := TRUE;
   #Sts.Pusher.UsedInRightPos := TRUE;

   #COut.PusherHoriz.AllStandstill := TRUE;
   #COut.PusherHoriz.Left_CheckNext := FALSE;
   #COut.PusherHoriz.Right_CheckNext := FALSE;

   FOR #i := 1 TO "MAX_PUSHER" DO

       #PusherHoriz[#i].Cin.Manager.EnableStopDoorOpeningReq := #CIn.Manager.EnableStopDoorOpeningReq;
       #PusherHoriz[#i].Cin.Manager.EnableStopInPhase := #Ctrl.StopInPhase;
       #PusherHoriz[#i].Cin.Manager.EnableStopProgrammed := #Ctrl.StopProgrammed;

       #PusherHoriz[#i].Cin.Manager.Control_ON := #Ctrl.Pusher.Aut_Left OR #Ctrl.Pusher.Aut_Right OR #Ctrl.Pusher.Man_Left OR #Ctrl.Pusher.Man_Right;
       #PusherHoriz[#i].Cin.Manager.Work := (#Ctrl.Pusher.Aut_Right AND (#Sts.Pusher.Used[#i] OR #Sts.Pusher.AllDown) AND NOT #Ctrl.StopInPhase AND NOT #Ctrl.StopProgrammed) OR #Ctrl.Pusher.Man_Right;
       #PusherHoriz[#i].Cin.Manager.Rest := (#Ctrl.Pusher.Aut_Left  AND (#Sts.Pusher.Used[#i] OR #Sts.Pusher.AllDown) AND NOT #Ctrl.StopInPhase AND NOT #Ctrl.StopProgrammed) OR #Ctrl.Pusher.Man_Left;

       #PusherHoriz[#i].Cin.Rest_ExtEnable := (#AreaInterface.Man AND NOT #Sts.Semiautomatic AND #Sts.OP_CanMoveFreely) OR (#PusherHoriz[#i].Cin.Manager.Control_ON AND #Sts.Pusher.Used[#i]) OR #Sts.Pusher.AllDown;
       #PusherHoriz[#i].Cin.Work_ExtEnable := #PusherHoriz[#i].Cin.Rest_ExtEnable;
       #PusherHoriz[#i].Cin.ExternalAlarms := FALSE;


       #PusherHoriz[#i](AreaInterface := #AreaInterface,
                        ZSI := #ZSI,
                        DSI := #DSI.PusherHoriz,
                        Config := #Config.PusherHoriz[#i],
                        Alarm := #Alarm.PusherHoriz[#i],
                        Warning := #Warning.PusherHoriz[#i]);

       IF NOT #PusherHoriz[#i].COut.Rest THEN
           #Sts.Pusher.InLeftPos := FALSE;
       END_IF;
       IF NOT #PusherHoriz[#i].COut.Work THEN
           #Sts.Pusher.InRightPos := FALSE;
       END_IF;
       IF #Sts.Pusher.Used[#i] AND
           NOT #PusherHoriz[#i].COut.Rest
       THEN
           #Sts.Pusher.UsedInLeftPos := FALSE;
       END_IF;
       IF #Sts.Pusher.Used[#i] AND
           NOT #PusherHoriz[#i].COut.Work
       THEN
           #Sts.Pusher.UsedInRightPos := FALSE;
       END_IF;

       IF NOT #PusherHoriz[#i].COut.Standstill THEN
           #COut.PusherHoriz.AllStandstill := FALSE;
       END_IF;

       IF #PusherHoriz[#i].COut.Rest_CheckNext THEN
           #COut.PusherHoriz.Left_CheckNext := TRUE;
       END_IF;
       IF #PusherHoriz[#i].COut.Work_CheckNext THEN
           #COut.PusherHoriz.Right_CheckNext := TRUE;
       END_IF;

       IF #i= 1 THEN
           #PusherHoriz_MachineInterface := #PusherHoriz[#i].MachineInterface;
       ELSE
           #PusherHoriz_MachineInterface := "MachineInterface_2_To_1"(MachineInterface_1 := #PusherHoriz_MachineInterface,
                                                                      MachineInterface_2 := #PusherHoriz[#i].MachineInterface,
                                                                      AdditionalAlarms := FALSE,
                                                                      AdditionalWarnings := FALSE);
       END_IF;
   END_FOR;

   #COut.PusherHoriz.InLeftPos := #Sts.Pusher.InLeftPos;
   #COut.PusherHoriz.InRightPos := #Sts.Pusher.InRightPos;
END_REGION

REGION Network 78: At Rest / At work positive/negative edge
   RUNG wire#powerrail
      P_Contact(operand := #PusherHoriz[1].COut.Rest, bit := #AUX.PusherHoriz_InLeftPos)
      Coil( #PE.PusherHoriz_InLeftPos )
   END_RUNG
   RUNG wire#powerrail
      P_Contact(operand := #PusherHoriz[1].COut.Work, bit := #AUX.PusherHoriz_InRightPos)
      Coil( #PE.PusherHoriz_InRightPos )
   END_RUNG
   // the same network as SCL:
   #_w1 := #PusherHoriz[1].COut.Rest AND NOT #AUX.PusherHoriz_InLeftPos;   // rising edge of #PusherHoriz[1].COut.Rest
   #AUX.PusherHoriz_InLeftPos := #PusherHoriz[1].COut.Rest;
   #PE.PusherHoriz_InLeftPos := #_w1;
   #_w2 := #PusherHoriz[1].COut.Work AND NOT #AUX.PusherHoriz_InRightPos;   // rising edge of #PusherHoriz[1].COut.Work
   #AUX.PusherHoriz_InRightPos := #PusherHoriz[1].COut.Work;
   #PE.PusherHoriz_InRightPos := #_w2;
END_REGION

REGION Network 79: Rest to work time calculation
   RUNG wire#powerrail
      Contact( #PusherHoriz[1].DataOut.WorkSolenoid )
      I_Contact( #Sts.CycleTime.PusherHoriz.R_To_W_Exe )
      { S7_Templates := "date_type := DTL" } RD_SYS_T(RET_VAL => #ReturnVal, OUT => #Sts.CycleTime.PusherHoriz.DT_W_Start)
      S_Coil( #Sts.CycleTime.PusherHoriz.R_To_W_Exe )
   END_RUNG
   RUNG wire#powerrail
      Contact( #Sts.CycleTime.PusherHoriz.R_To_W_Exe )
      wire#w1
      Contact( #PE.PusherHoriz_InRightPos )
      wire#w2
      { S7_Templates := "date_type := DTL" } RD_SYS_T(RET_VAL => #ReturnVal, OUT => #Sts.CycleTime.PusherHoriz.DT_W_Stop)
   END_RUNG
   RUNG wire#w1
      I_Contact( #PusherHoriz[1].DataOut.WorkSolenoid )
   END_RUNG wire#w2
   RUNG wire#w2
      { S7_Templates := "[date_type := DTL, time_type := Time]" } T_DIFF(IN1 := #Sts.CycleTime.PusherHoriz.DT_W_Stop, IN2 := #Sts.CycleTime.PusherHoriz.DT_W_Start, OUT => #HMI.PusherHoriz.Last_R_to_W_Time)
   END_RUNG
   RUNG wire#w2
      Add(in1 := #HMI.PusherHoriz.Buffer_R_to_W_Time[1].ID, in2 := 1, out => #HMI.PusherHoriz.Last_R_to_W_ID)
   END_RUNG
   RUNG wire#powerrail
      Contact( #Sts.CycleTime.PusherHoriz.R_To_W_Exe )
      I_Contact( #PusherHoriz[1].DataOut.WorkSolenoid )
      R_Coil( #Sts.CycleTime.PusherHoriz.R_To_W_Exe )
   END_RUNG
   // the same network as SCL:
   #ReturnVal := RD_SYS_T(EN := #PusherHoriz[1].DataOut.WorkSolenoid AND NOT #Sts.CycleTime.PusherHoriz.R_To_W_Exe,
                          OUT => #Sts.CycleTime.PusherHoriz.DT_W_Start,
                          ENO => #_w1);
   IF #_w1 THEN #Sts.CycleTime.PusherHoriz.R_To_W_Exe := TRUE; END_IF;
   IF #Sts.CycleTime.PusherHoriz.R_To_W_Exe AND (#PE.PusherHoriz_InRightPos OR NOT #PusherHoriz[1].DataOut.WorkSolenoid) THEN
       #ReturnVal := RD_SYS_T(OUT => #Sts.CycleTime.PusherHoriz.DT_W_Stop);
       T_DIFF(IN1 := #Sts.CycleTime.PusherHoriz.DT_W_Stop,
              IN2 := #Sts.CycleTime.PusherHoriz.DT_W_Start,
              OUT => #HMI.PusherHoriz.Last_R_to_W_Time);
       #HMI.PusherHoriz.Last_R_to_W_ID := #HMI.PusherHoriz.Buffer_R_to_W_Time[1].ID + 1;
   END_IF;
   IF #Sts.CycleTime.PusherHoriz.R_To_W_Exe AND NOT #PusherHoriz[1].DataOut.WorkSolenoid THEN
       #Sts.CycleTime.PusherHoriz.R_To_W_Exe := FALSE;
   END_IF;
END_REGION

REGION Network 80: Work to rest time calculation
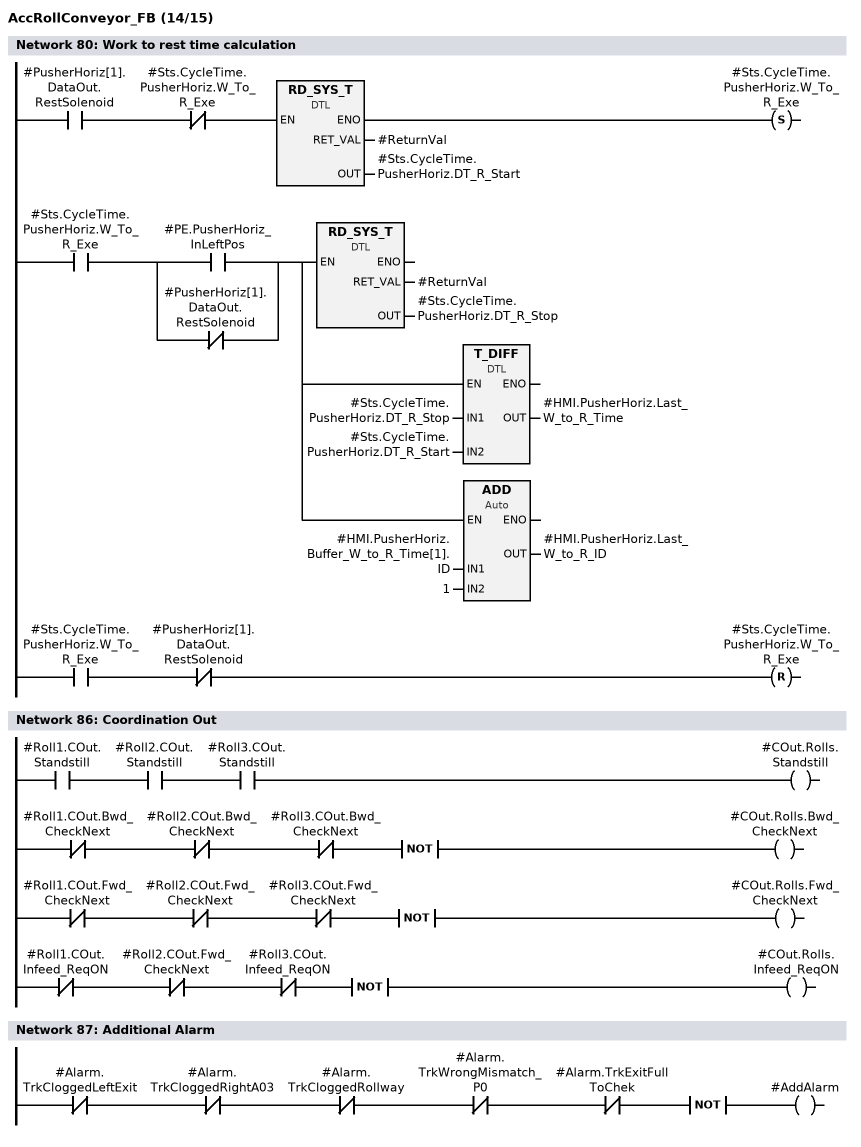
   RUNG wire#powerrail
      Contact( #PusherHoriz[1].DataOut.RestSolenoid )
      I_Contact( #Sts.CycleTime.PusherHoriz.W_To_R_Exe )
      { S7_Templates := "date_type := DTL" } RD_SYS_T(RET_VAL => #ReturnVal, OUT => #Sts.CycleTime.PusherHoriz.DT_R_Start)
      S_Coil( #Sts.CycleTime.PusherHoriz.W_To_R_Exe )
   END_RUNG
   RUNG wire#powerrail
      Contact( #Sts.CycleTime.PusherHoriz.W_To_R_Exe )
      wire#w1
      Contact( #PE.PusherHoriz_InLeftPos )
      wire#w2
      { S7_Templates := "date_type := DTL" } RD_SYS_T(RET_VAL => #ReturnVal, OUT => #Sts.CycleTime.PusherHoriz.DT_R_Stop)
   END_RUNG
   RUNG wire#w1
      I_Contact( #PusherHoriz[1].DataOut.RestSolenoid )
   END_RUNG wire#w2
   RUNG wire#w2
      { S7_Templates := "[date_type := DTL, time_type := Time]" } T_DIFF(IN1 := #Sts.CycleTime.PusherHoriz.DT_R_Stop, IN2 := #Sts.CycleTime.PusherHoriz.DT_R_Start, OUT => #HMI.PusherHoriz.Last_W_to_R_Time)
   END_RUNG
   RUNG wire#w2
      Add(in1 := #HMI.PusherHoriz.Buffer_W_to_R_Time[1].ID, in2 := 1, out => #HMI.PusherHoriz.Last_W_to_R_ID)
   END_RUNG
   RUNG wire#powerrail
      Contact( #Sts.CycleTime.PusherHoriz.W_To_R_Exe )
      I_Contact( #PusherHoriz[1].DataOut.RestSolenoid )
      R_Coil( #Sts.CycleTime.PusherHoriz.W_To_R_Exe )
   END_RUNG
   // the same network as SCL:
   #ReturnVal := RD_SYS_T(EN := #PusherHoriz[1].DataOut.RestSolenoid AND NOT #Sts.CycleTime.PusherHoriz.W_To_R_Exe,
                          OUT => #Sts.CycleTime.PusherHoriz.DT_R_Start,
                          ENO => #_w1);
   IF #_w1 THEN #Sts.CycleTime.PusherHoriz.W_To_R_Exe := TRUE; END_IF;
   IF #Sts.CycleTime.PusherHoriz.W_To_R_Exe AND (#PE.PusherHoriz_InLeftPos OR NOT #PusherHoriz[1].DataOut.RestSolenoid) THEN
       #ReturnVal := RD_SYS_T(OUT => #Sts.CycleTime.PusherHoriz.DT_R_Stop);
       T_DIFF(IN1 := #Sts.CycleTime.PusherHoriz.DT_R_Stop,
              IN2 := #Sts.CycleTime.PusherHoriz.DT_R_Start,
              OUT => #HMI.PusherHoriz.Last_W_to_R_Time);
       #HMI.PusherHoriz.Last_W_to_R_ID := #HMI.PusherHoriz.Buffer_W_to_R_Time[1].ID + 1;
   END_IF;
   IF #Sts.CycleTime.PusherHoriz.W_To_R_Exe AND NOT #PusherHoriz[1].DataOut.RestSolenoid THEN
       #Sts.CycleTime.PusherHoriz.W_To_R_Exe := FALSE;
   END_IF;
END_REGION

REGION Network 81 (SCL): Init buffers & average calculations
   IF "PPrf_MAIN".ON_WORK.Header.PrgNo <> #Sts.CycleTime.PPrf_PrgNoSave OR "PPrf_MAIN".ON_WORK.Header.PrgNo <= 0 THEN

       FOR #i := 1 TO #BUFFER_ITEMS DO
           #HMI.PusherHoriz.Buffer_R_to_W_Time[#i].ID := 0;
           #HMI.PusherHoriz.Buffer_R_to_W_Time[#i].Value := T#0s;
           #HMI.PusherHoriz.Buffer_W_to_R_Time[#i].ID := 0;
           #HMI.PusherHoriz.Buffer_W_to_R_Time[#i].Value := T#0s;
       END_FOR;

       #HMI.PusherHoriz.Last_R_to_W_ID := 0;
       #HMI.PusherHoriz.Last_R_to_W_Time := T#0ms;
       #HMI.PusherHoriz.Avg_R_to_W_Time := #Config.PusherHoriz[1].V.WorkTimeOut;
       #HMI.PusherHoriz.Last_W_to_R_ID := 0;
       #HMI.PusherHoriz.Last_W_to_R_Time := T#0ms;
       #HMI.PusherHoriz.Avg_W_to_R_Time := #Config.PusherHoriz[1].V.RestTimeOut;

   END_IF;


   #Sts.CycleTime.PPrf_PrgNoSave := "PPrf_MAIN".ON_WORK.Header.PrgNo ;
END_REGION

REGION Network 82 (SCL): Add new items to Rest-TO-Work buffer & calculate average

   IF #HMI.PusherHoriz.Last_R_to_W_Time >= #Config.PusherHoriz[1].V.WorkTimeOut OR #Alarm.PusherHoriz[1].TimeOutWork THEN

       #HMI.PusherHoriz.Last_R_to_W_ID := -1; // Force red background on the HMI visualization



   ELSIF #HMI.PusherHoriz.Last_R_to_W_ID <> #HMI.PusherHoriz.Buffer_R_to_W_Time[1].ID AND #HMI.PusherHoriz.Last_R_to_W_Time < #Config.PusherHoriz[1].V.WorkTimeOut AND #HMI.PusherHoriz.Last_R_to_W_Time > T#0ms THEN

       #i := #BUFFER_ITEMS;

       WHILE #i >= 2 DO

           #HMI.PusherHoriz.Buffer_R_to_W_Time[#i] := #HMI.PusherHoriz.Buffer_R_to_W_Time[#i - 1];

           #i -= 1;

       END_WHILE;

       #HMI.PusherHoriz.Buffer_R_to_W_Time[1].ID := #HMI.PusherHoriz.Last_R_to_W_ID;
       #HMI.PusherHoriz.Buffer_R_to_W_Time[1].Value := #HMI.PusherHoriz.Last_R_to_W_Time;

       #Sts.CycleTime.PusherHoriz.R_To_W_Items := 0;
       #Sts.CycleTime.PusherHoriz.R_To_W_Sum := T#0s;


       FOR #i := 1 TO #BUFFER_ITEMS DO

           IF #HMI.PusherHoriz.Buffer_R_to_W_Time[#i].ID > 0 AND #HMI.PusherHoriz.Buffer_R_to_W_Time[#i].Value > T#0ms THEN
               #Sts.CycleTime.PusherHoriz.R_To_W_Items += 1;
               #Sts.CycleTime.PusherHoriz.R_To_W_Sum := #Sts.CycleTime.PusherHoriz.R_To_W_Sum + #HMI.PusherHoriz.Buffer_R_to_W_Time[#i].Value;
           END_IF;

       END_FOR;

       IF #Sts.CycleTime.PusherHoriz.R_To_W_Items >= 5 THEN
           #HMI.PusherHoriz.Avg_R_to_W_Time := #Sts.CycleTime.PusherHoriz.R_To_W_Sum / #Sts.CycleTime.PusherHoriz.R_To_W_Items;
       ELSE
           #HMI.PusherHoriz.Avg_R_to_W_Time := #Config.PusherHoriz[1].V.WorkTimeOut;
       END_IF;

   END_IF;


   //#HMI.PusherHoriz.Avg_CycleTime_S := DINT_TO_LREAL(TIME_TO_DINT(((#HMI.PusherHoriz.Avg_R_to_W_Time + #HMI.PusherHoriz.Avg_W_to_R_Time) / 2))) / 1000;

   #HMI.PusherHoriz.Avg_CycleTime_S := DINT_TO_LREAL(TIME_TO_DINT(#HMI.PusherHoriz.Avg_R_to_W_Time)) / 1000;
END_REGION

REGION Network 83 (SCL): Add new items to Work-TO-Rest buffer & calculate average
   IF #HMI.PusherHoriz.Last_W_to_R_Time >= #Config.PusherHoriz[1].V.RestTimeOut OR #Alarm.PusherHoriz[1].TimeOutRest THEN

       #HMI.PusherHoriz.Last_W_to_R_ID := -1; // Force red background on the HMI visualization

   ELSIF #HMI.PusherHoriz.Last_W_to_R_ID <> #HMI.PusherHoriz.Buffer_W_to_R_Time[1].ID AND #HMI.PusherHoriz.Last_W_to_R_Time < #Config.PusherHoriz[1].V.RestTimeOut AND #HMI.PusherHoriz.Last_W_to_R_Time > T#0ms  THEN

       #i := #BUFFER_ITEMS;

       WHILE #i >= 2 DO

           #HMI.PusherHoriz.Buffer_W_to_R_Time[#i] := #HMI.PusherHoriz.Buffer_W_to_R_Time[#i - 1];

           #i -= 1;

       END_WHILE;

       #HMI.PusherHoriz.Buffer_W_to_R_Time[1].ID := #HMI.PusherHoriz.Last_W_to_R_ID;
       #HMI.PusherHoriz.Buffer_W_to_R_Time[1].Value := #HMI.PusherHoriz.Last_W_to_R_Time;

       #Sts.CycleTime.PusherHoriz.W_To_R_Items := 0;
       #Sts.CycleTime.PusherHoriz.W_To_R_Sum := T#0s;


       FOR #i := 1 TO #BUFFER_ITEMS DO

           IF #HMI.PusherHoriz.Buffer_W_to_R_Time[#i].ID > 0 AND #HMI.PusherHoriz.Buffer_W_to_R_Time[#i].Value > T#0ms  THEN
               #Sts.CycleTime.PusherHoriz.W_To_R_Items += 1;
               #Sts.CycleTime.PusherHoriz.W_To_R_Sum := #Sts.CycleTime.PusherHoriz.W_To_R_Sum + #HMI.PusherHoriz.Buffer_W_to_R_Time[#i].Value;
           END_IF;

       END_FOR;

       IF #Sts.CycleTime.PusherHoriz.W_To_R_Items >= 5 THEN
           #HMI.PusherHoriz.Avg_W_to_R_Time := #Sts.CycleTime.PusherHoriz.W_To_R_Sum / #Sts.CycleTime.PusherHoriz.W_To_R_Items;
       ELSE
           #HMI.PusherHoriz.Avg_W_to_R_Time := #Config.PusherHoriz[1].V.RestTimeOut;
       END_IF;

   END_IF;
END_REGION

REGION Network 84: >
END_REGION

REGION Network 85: <<< MACHINE STATUS >>>
END_REGION

REGION Network 86: Coordination Out
   RUNG wire#powerrail
      Contact( #Roll1.COut.Standstill )
      Contact( #Roll2.COut.Standstill )
      Contact( #Roll3.COut.Standstill )
      Coil( #COut.Rolls.Standstill )
   END_RUNG
   RUNG wire#powerrail
      I_Contact( #Roll1.COut.Bwd_CheckNext )
      I_Contact( #Roll2.COut.Bwd_CheckNext )
      I_Contact( #Roll3.COut.Bwd_CheckNext )
      Not()
      Coil( #COut.Rolls.Bwd_CheckNext )
   END_RUNG
   RUNG wire#powerrail
      I_Contact( #Roll1.COut.Fwd_CheckNext )
      I_Contact( #Roll2.COut.Fwd_CheckNext )
      I_Contact( #Roll3.COut.Fwd_CheckNext )
      Not()
      Coil( #COut.Rolls.Fwd_CheckNext )
   END_RUNG
   RUNG wire#powerrail
      I_Contact( #Roll1.COut.Infeed_ReqON )
      I_Contact( #Roll2.COut.Fwd_CheckNext )
      I_Contact( #Roll3.COut.Infeed_ReqON )
      Not()
      Coil( #COut.Rolls.Infeed_ReqON )
   END_RUNG
   // the same network as SCL:
   #COut.Rolls.Standstill := #Roll1.COut.Standstill AND #Roll2.COut.Standstill AND #Roll3.COut.Standstill;
   #COut.Rolls.Bwd_CheckNext := NOT (NOT #Roll1.COut.Bwd_CheckNext AND NOT #Roll2.COut.Bwd_CheckNext AND NOT #Roll3.COut.Bwd_CheckNext);
   #COut.Rolls.Fwd_CheckNext := NOT (NOT #Roll1.COut.Fwd_CheckNext AND NOT #Roll2.COut.Fwd_CheckNext AND NOT #Roll3.COut.Fwd_CheckNext);
   #COut.Rolls.Infeed_ReqON := NOT (NOT #Roll1.COut.Infeed_ReqON AND NOT #Roll2.COut.Fwd_CheckNext AND NOT #Roll3.COut.Infeed_ReqON);
END_REGION

REGION Network 87: Additional Alarm
   RUNG wire#powerrail
      I_Contact( #Alarm.TrkCloggedLeftExit )
      I_Contact( #Alarm.TrkCloggedRightA03 )
      I_Contact( #Alarm.TrkCloggedRollway )
      I_Contact( #Alarm.TrkWrongMismatch_P0 )
      I_Contact( #Alarm.TrkExitFullToChek )
      Not()
      Coil( #AddAlarm )
   END_RUNG
   // the same network as SCL:
   #AddAlarm := NOT (NOT #Alarm.TrkCloggedLeftExit AND NOT #Alarm.TrkCloggedRightA03 AND NOT #Alarm.TrkCloggedRollway AND NOT #Alarm.TrkWrongMismatch_P0 AND NOT #Alarm.TrkExitFullToChek);
END_REGION

REGION Network 88: Collect machine to zone interface (internal machines OR)
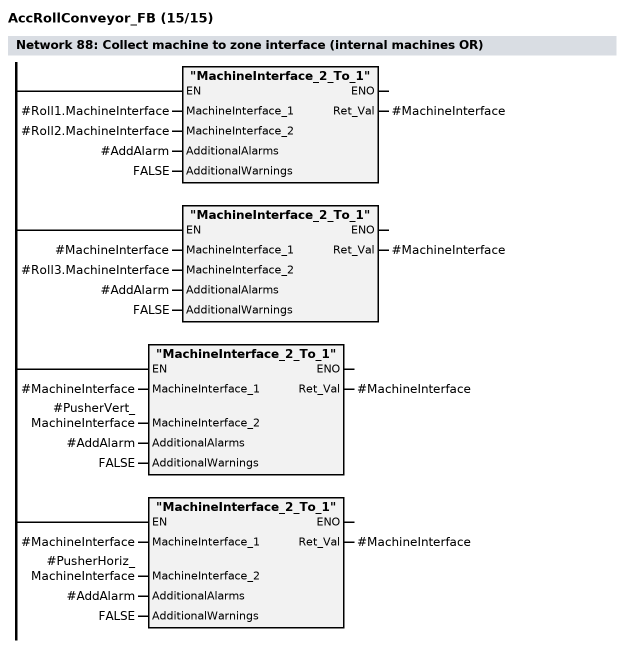
   RUNG wire#powerrail
      "MachineInterface_2_To_1"(MachineInterface_1 := #Roll1.MachineInterface, MachineInterface_2 := #Roll2.MachineInterface, AdditionalAlarms := #AddAlarm, AdditionalWarnings := FALSE, Ret_Val => #MachineInterface)
   END_RUNG
   RUNG wire#powerrail
      "MachineInterface_2_To_1"(MachineInterface_1 := #MachineInterface, MachineInterface_2 := #Roll3.MachineInterface, AdditionalAlarms := #AddAlarm, AdditionalWarnings := FALSE, Ret_Val => #MachineInterface)
   END_RUNG
   RUNG wire#powerrail
      "MachineInterface_2_To_1"(MachineInterface_1 := #MachineInterface, MachineInterface_2 := #PusherVert_MachineInterface, AdditionalAlarms := #AddAlarm, AdditionalWarnings := FALSE, Ret_Val => #MachineInterface)
   END_RUNG
   RUNG wire#powerrail
      "MachineInterface_2_To_1"(MachineInterface_1 := #MachineInterface, MachineInterface_2 := #PusherHoriz_MachineInterface, AdditionalAlarms := #AddAlarm, AdditionalWarnings := FALSE, Ret_Val => #MachineInterface)
   END_RUNG
   // the same network as SCL:
   #MachineInterface := "MachineInterface_2_To_1"(MachineInterface_1 := #Roll1.MachineInterface,
                           MachineInterface_2 := #Roll2.MachineInterface,
                           AdditionalAlarms := #AddAlarm,
                           AdditionalWarnings := FALSE);
   #MachineInterface := "MachineInterface_2_To_1"(MachineInterface_1 := #MachineInterface,
                           MachineInterface_2 := #Roll3.MachineInterface,
                           AdditionalAlarms := #AddAlarm,
                           AdditionalWarnings := FALSE);
   #MachineInterface := "MachineInterface_2_To_1"(MachineInterface_1 := #MachineInterface,
                           MachineInterface_2 := #PusherVert_MachineInterface,
                           AdditionalAlarms := #AddAlarm,
                           AdditionalWarnings := FALSE);
   #MachineInterface := "MachineInterface_2_To_1"(MachineInterface_1 := #MachineInterface,
                           MachineInterface_2 := #PusherHoriz_MachineInterface,
                           AdditionalAlarms := #AddAlarm,
                           AdditionalWarnings := FALSE);
END_REGION

REGION Network 89 (SCL): Ack stop in phase and stop programmed

   #MachineInterface.AckStopInPhase := #MachineInterface.AckStopInPhase AND (#COut.Manager.Empty OR #MachineInterface.Aborting);
   #MachineInterface.AckStopProgrammed := #MachineInterface.AckStopInPhase AND(#COut.Manager.Empty OR #MachineInterface.Aborting);
END_REGION

REGION Network 90: >
END_REGION

REGION Network 91: >
END_REGION
END_FUNCTION_BLOCK
